    |   movel([0.036971, -1.567857, -2.417169, -0.727363, 1.570796, 1.607768],accel_mss,speed_ms,0,blend_radius_m)
    |   movel([0.032034, -1.570539, -2.414494, -0.727356, 1.570796, 1.602831],accel_mss,speed_ms,0,blend_radius_m)
    |   movel([0.033488, -1.569504, -2.415528, -0.727358, 1.570796, 1.604284],accel_mss,speed_ms,0,blend_radius_m)
    |   movel([0.034915, -1.568368, -2.416660, -0.727361, 1.570796, 1.605712],accel_mss,speed_ms,0,blend_radius_m)
    |   movel([0.036304, -1.567153, -2.417869, -0.727367, 1.570796, 1.607100],accel_mss,speed_ms,0,blend_radius_m)
    |   movel([0.037649, -1.565876, -2.419138, -0.727376, 1.570796, 1.608445],accel_mss,speed_ms,0,blend_radius_m)
    |   movel([0.040174, -1.563204, -2.421782, -0.727403, 1.570796, 1.610970],accel_mss,speed_ms,0,blend_radius_m)
    |   movel([0.042420, -1.560504, -2.424443, -0.727442, 1.570796, 1.613216],accel_mss,speed_ms,0,blend_radius_m)
    |   movel([0.044692, -1.557524, -2.427367, -0.727498, 1.570796, 1.615489],accel_mss,speed_ms,0,blend_radius_m)
    |   movel([0.046838, -1.554469, -2.430349, -0.727571, 1.570796, 1.617635],accel_mss,speed_ms,0,blend_radius_m)
    |   movel([0.047827, -1.552916, -2.431859, -0.727614, 1.570796, 1.618623],accel_mss,speed_ms,0,blend_radius_m)
    |   movel([0.048742, -1.551347, -2.433381, -0.727661, 1.570796, 1.619539],accel_mss,speed_ms,0,blend_radius_m)
    |   movel([0.049567, -1.549765, -2.434911, -0.727713, 1.570796, 1.620363],accel_mss,speed_ms,0,blend_radius_m)
    |   movel([0.050288, -1.548168, -2.436452, -0.727769, 1.570796, 1.621084],accel_mss,speed_ms,0,blend_radius_m)
    |   movel([0.050654, -1.547170, -2.437413, -0.727806, 1.570796, 1.621451],accel_mss,speed_ms,0,blend_radius_m)
    |   movel([0.050929, -1.546167, -2.438377, -0.727845, 1.570796, 1.621725],accel_mss,speed_ms,0,blend_radius_m)
    |   movel([0.051225, -1.544162, -2.440299, -0.727928, 1.570796, 1.622021],accel_mss,speed_ms,0,blend_radius_m)
    |   movel([0.051211, -1.542184, -2.442189, -0.728016, 1.570796, 1.622007],accel_mss,speed_ms,0,blend_radius_m)
    |   movel([0.050919, -1.540264, -2.444018, -0.728108, 1.570796, 1.621716],accel_mss,speed_ms,0,blend_radius_m)
    |   movel([0.050389, -1.538428, -2.445760, -0.728201, 1.570796, 1.621186],accel_mss,speed_ms,0,blend_radius_m)
    |   movel([0.049659, -1.536708, -2.447388, -0.728293, 1.570796, 1.620455],accel_mss,speed_ms,0,blend_radius_m)
    |   movel([0.048760, -1.535134, -2.448874, -0.728381, 1.570796, 1.619557],accel_mss,speed_ms,0,blend_radius_m)
    |   movel([0.047734, -1.533734, -2.450192, -0.728463, 1.570796, 1.618531],accel_mss,speed_ms,0,blend_radius_m)
    |   movel([0.046969, -1.533087, -2.450800, -0.728502, 1.570796, 1.617766],accel_mss,speed_ms,0,blend_radius_m)
    |   movel([0.046036, -1.532733, -2.451133, -0.728524, 1.570796, 1.616832],accel_mss,speed_ms,0,blend_radius_m)
    |   movel([0.044989, -1.532658, -2.451202, -0.728528, 1.570796, 1.615785],accel_mss,speed_ms,0,blend_radius_m)
    |   movel([0.043886, -1.532851, -2.451022, -0.728516, 1.570796, 1.614683],accel_mss,speed_ms,0,blend_radius_m)
    |   movel([0.042779, -1.533292, -2.450607, -0.728490, 1.570796, 1.613575],accel_mss,speed_ms,0,blend_radius_m)
    |   movel([0.041722, -1.533971, -2.449969, -0.728449, 1.570796, 1.612519],accel_mss,speed_ms,0,blend_radius_m)
    |   movel([0.040776, -1.534867, -2.449125, -0.728396, 1.570796, 1.611572],accel_mss,speed_ms,0,blend_radius_m)
    |   movel([0.039990, -1.535966, -2.448089, -0.728334, 1.570796, 1.610787],accel_mss,speed_ms,0,blend_radius_m)
    |   movel([0.038953, -1.537691, -2.446459, -0.728239, 1.570796, 1.609749],accel_mss,speed_ms,0,blend_radius_m)
    |   movel([0.037826, -1.539382, -2.444855, -0.728152, 1.570796, 1.608622],accel_mss,speed_ms,0,blend_radius_m)
    |   movel([0.036599, -1.541021, -2.443297, -0.728071, 1.570796, 1.607395],accel_mss,speed_ms,0,blend_radius_m)
    |   movel([0.035257, -1.542593, -2.441799, -0.727997, 1.570796, 1.606053],accel_mss,speed_ms,0,blend_radius_m)
    |   movel([0.033791, -1.544077, -2.440380, -0.727932, 1.570796, 1.604587],accel_mss,speed_ms,0,blend_radius_m)
    |   movel([0.032187, -1.545460, -2.439055, -0.727874, 1.570796, 1.602984],accel_mss,speed_ms,0,blend_radius_m)
    |   movel([0.030433, -1.546725, -2.437841, -0.727823, 1.570796, 1.601229],accel_mss,speed_ms,0,blend_radius_m)
    |   movel([0.028519, -1.547854, -2.436755, -0.727781, 1.570796, 1.599315],accel_mss,speed_ms,0,blend_radius_m)
    |   movel([0.027475, -1.548332, -2.436294, -0.727763, 1.570796, 1.598272],accel_mss,speed_ms,0,blend_radius_m)
    |   movel([0.026412, -1.548698, -2.435941, -0.727750, 1.570796, 1.597208],accel_mss,speed_ms,0,blend_radius_m)
    |   movel([0.024268, -1.549225, -2.435433, -0.727731, 1.570796, 1.595065],accel_mss,speed_ms,0,blend_radius_m)
    |   movel([0.022596, -1.549491, -2.435176, -0.727722, 1.570796, 1.593392],accel_mss,speed_ms,0,blend_radius_m)
    |   movel([0.021010, -1.549563, -2.435106, -0.727720, 1.570796, 1.591806],accel_mss,speed_ms,0,blend_radius_m)
    |   movel([0.019511, -1.549457, -2.435209, -0.727723, 1.570796, 1.590308],accel_mss,speed_ms,0,blend_radius_m)
    |   movel([0.018095, -1.549187, -2.435470, -0.727733, 1.570796, 1.588891],accel_mss,speed_ms,0,blend_radius_m)
    |   movel([0.016758, -1.548771, -2.435871, -0.727747, 1.570796, 1.587554],accel_mss,speed_ms,0,blend_radius_m)
    |   movel([0.015496, -1.548222, -2.436399, -0.727767, 1.570796, 1.586293],accel_mss,speed_ms,0,blend_radius_m)
    |   movel([0.014313, -1.547556, -2.437041, -0.727792, 1.570796, 1.585109],accel_mss,speed_ms,0,blend_radius_m)
    |   movel([0.013202, -1.546790, -2.437779, -0.727821, 1.570796, 1.583999],accel_mss,speed_ms,0,blend_radius_m)
    |   movel([0.012162, -1.545938, -2.438597, -0.727854, 1.570796, 1.582959],accel_mss,speed_ms,0,blend_radius_m)
    |   movel([0.011193, -1.545012, -2.439485, -0.727892, 1.570796, 1.581989],accel_mss,speed_ms,0,blend_radius_m)
    |   movel([0.009457, -1.543013, -2.441397, -0.727978, 1.570796, 1.580253],accel_mss,speed_ms,0,blend_radius_m)
    |   movel([0.007979, -1.540912, -2.443401, -0.728076, 1.570796, 1.578775],accel_mss,speed_ms,0,blend_radius_m)
    |   movel([0.006747, -1.538836, -2.445373, -0.728179, 1.570796, 1.577544],accel_mss,speed_ms,0,blend_radius_m)
    |   movel([0.005914, -1.537189, -2.446933, -0.728266, 1.570796, 1.576710],accel_mss,speed_ms,0,blend_radius_m)
    |   movel([0.005168, -1.535434, -2.448591, -0.728364, 1.570796, 1.575964],accel_mss,speed_ms,0,blend_radius_m)
    |   movel([0.004519, -1.533579, -2.450338, -0.728472, 1.570796, 1.575315],accel_mss,speed_ms,0,blend_radius_m)
    |   movel([0.003986, -1.531636, -2.452161, -0.728592, 1.570796, 1.574783],accel_mss,speed_ms,0,blend_radius_m)
    |   movel([0.003580, -1.529616, -2.454051, -0.728722, 1.570796, 1.574376],accel_mss,speed_ms,0,blend_radius_m)
    |   movel([0.003317, -1.527529, -2.455996, -0.728864, 1.570796, 1.574114],accel_mss,speed_ms,0,blend_radius_m)
    |   movel([0.003214, -1.525386, -2.457986, -0.729017, 1.570796, 1.574010],accel_mss,speed_ms,0,blend_radius_m)
    |   movel([0.003284, -1.523198, -2.460010, -0.729181, 1.570796, 1.574081],accel_mss,speed_ms,0,blend_radius_m)
    |   movel([0.003542, -1.520975, -2.462059, -0.729355, 1.570796, 1.574338],accel_mss,speed_ms,0,blend_radius_m)
    |   movel([0.004003, -1.518731, -2.464119, -0.729539, 1.570796, 1.574800],accel_mss,speed_ms,0,blend_radius_m)
    |   movel([0.004683, -1.516473, -2.466184, -0.729732, 1.570796, 1.575479],accel_mss,speed_ms,0,blend_radius_m)
    |   movel([0.005599, -1.514215, -2.468241, -0.729933, 1.570796, 1.576396],accel_mss,speed_ms,0,blend_radius_m)
    |   movel([0.006765, -1.511969, -2.470278, -0.730141, 1.570796, 1.577561],accel_mss,speed_ms,0,blend_radius_m)
    |   movel([0.008199, -1.509745, -2.472288, -0.730356, 1.570796, 1.578995],accel_mss,speed_ms,0,blend_radius_m)
    |   movel([0.009913, -1.507560, -2.474255, -0.730574, 1.570796, 1.580709],accel_mss,speed_ms,0,blend_radius_m)
    |   movel([0.011923, -1.505424, -2.476171, -0.730794, 1.570796, 1.582720],accel_mss,speed_ms,0,blend_radius_m)
    |   movel([0.012797, -1.504654, -2.476860, -0.730876, 1.570796, 1.583593],accel_mss,speed_ms,0,blend_radius_m)
    |   movel([0.013277, -1.504331, -2.477148, -0.730910, 1.570796, 1.584073],accel_mss,speed_ms,0,blend_radius_m)
    |   movel([0.013789, -1.504089, -2.477364, -0.730936, 1.570796, 1.584585],accel_mss,speed_ms,0,blend_radius_m)
    |   movel([0.014561, -1.503942, -2.477496, -0.730952, 1.570796, 1.585357],accel_mss,speed_ms,0,blend_radius_m)
    |   movel([0.015250, -1.504040, -2.477408, -0.730941, 1.570796, 1.586046],accel_mss,speed_ms,0,blend_radius_m)
    |   movel([0.015830, -1.504330, -2.477149, -0.730910, 1.570796, 1.586626],accel_mss,speed_ms,0,blend_radius_m)
    |   movel([0.016270, -1.504757, -2.476767, -0.730865, 1.570796, 1.587067],accel_mss,speed_ms,0,blend_radius_m)
    |   movel([0.016900, -1.505930, -2.475718, -0.730741, 1.570796, 1.587696],accel_mss,speed_ms,0,blend_radius_m)
    |   movel([0.017252, -1.507271, -2.474515, -0.730603, 1.570796, 1.588049],accel_mss,speed_ms,0,blend_radius_m)
    |   movel([0.017654, -1.510076, -2.471990, -0.730323, 1.570796, 1.588450],accel_mss,speed_ms,0,blend_radius_m)
    |   movel([0.017877, -1.510551, -2.471561, -0.730277, 1.570796, 1.588673],accel_mss,speed_ms,0,blend_radius_m)
    |   movel([0.018117, -1.510629, -2.471491, -0.730270, 1.570796, 1.588914],accel_mss,speed_ms,0,blend_radius_m)
    |   movel([0.018485, -1.510569, -2.471544, -0.730275, 1.570796, 1.589281],accel_mss,speed_ms,0,blend_radius_m)
    |   movel([0.019067, -1.509442, -2.472562, -0.730385, 1.570796, 1.589864],accel_mss,speed_ms,0,blend_radius_m)
    |   movel([0.019568, -1.508284, -2.473604, -0.730501, 1.570796, 1.590365],accel_mss,speed_ms,0,blend_radius_m)
    |   movel([0.019982, -1.512436, -2.469855, -0.730098, 1.570796, 1.590778],accel_mss,speed_ms,0,blend_radius_m)
    |   movel([0.020558, -1.516505, -2.466155, -0.729729, 1.570796, 1.591354],accel_mss,speed_ms,0,blend_radius_m)
    |   movel([0.021295, -1.520487, -2.462508, -0.729394, 1.570796, 1.592091],accel_mss,speed_ms,0,blend_radius_m)
    |   movel([0.022191, -1.524383, -2.458915, -0.729091, 1.570796, 1.592987],accel_mss,speed_ms,0,blend_radius_m)
    |   movel([0.022649, -1.526045, -2.457375, -0.728969, 1.570796, 1.593445],accel_mss,speed_ms,0,blend_radius_m)
    |   movel([0.023296, -1.527701, -2.455836, -0.728852, 1.570796, 1.594092],accel_mss,speed_ms,0,blend_radius_m)
    |   movel([0.023724, -1.528467, -2.455122, -0.728800, 1.570796, 1.594520],accel_mss,speed_ms,0,blend_radius_m)
    |   movel([0.024238, -1.529159, -2.454478, -0.728753, 1.570796, 1.595035],accel_mss,speed_ms,0,blend_radius_m)
    |   movel([0.024855, -1.529751, -2.453924, -0.728713, 1.570796, 1.595651],accel_mss,speed_ms,0,blend_radius_m)
    |   movel([0.025587, -1.530219, -2.453487, -0.728683, 1.570796, 1.596384],accel_mss,speed_ms,0,blend_radius_m)
    |   movel([0.026170, -1.530452, -2.453270, -0.728668, 1.570796, 1.596966],accel_mss,speed_ms,0,blend_radius_m)
    |   movel([0.027457, -1.530642, -2.453092, -0.728655, 1.570796, 1.598253],accel_mss,speed_ms,0,blend_radius_m)
    |   movel([0.028149, -1.530613, -2.453119, -0.728657, 1.570796, 1.598945],accel_mss,speed_ms,0,blend_radius_m)
    |   movel([0.029599, -1.530339, -2.453375, -0.728675, 1.570796, 1.600395],accel_mss,speed_ms,0,blend_radius_m)
    |   movel([0.031098, -1.529820, -2.453860, -0.728709, 1.570796, 1.601894],accel_mss,speed_ms,0,blend_radius_m)
    |   movel([0.032596, -1.529109, -2.454524, -0.728756, 1.570796, 1.603392],accel_mss,speed_ms,0,blend_radius_m)
    |   movel([0.034042, -1.528253, -2.455322, -0.728814, 1.570796, 1.604839],accel_mss,speed_ms,0,blend_radius_m)
    |   movel([0.035389, -1.527306, -2.456203, -0.728880, 1.570796, 1.606186],accel_mss,speed_ms,0,blend_radius_m)
    |   movel([0.036582, -1.526318, -2.457121, -0.728950, 1.570796, 1.607378],accel_mss,speed_ms,0,blend_radius_m)
    |   speed_ms = 0.005
    |   movel([0.036582, -1.518669, -2.453733, -0.739987, 1.570796, 1.607378],accel_mss,speed_ms,0,blend_radius_m)
    |   speed_ms = 0.040
    |   movel([0.029707, -1.520999, -2.451592, -0.739798, 1.570796, 1.600503],accel_mss,speed_ms,0,blend_radius_m)
    |   speed_ms = 0.005
    |   movel([0.029707, -1.528629, -2.454972, -0.728789, 1.570796, 1.600503],accel_mss,speed_ms,0,blend_radius_m)
    |   speed_ms = 0.025
    |   movel([0.030662, -1.527790, -2.455753, -0.728846, 1.570796, 1.601458],accel_mss,speed_ms,0,blend_radius_m)
    |   movel([0.032483, -1.525887, -2.457521, -0.728981, 1.570796, 1.603279],accel_mss,speed_ms,0,blend_radius_m)
    |   movel([0.033332, -1.524844, -2.458488, -0.729057, 1.570796, 1.604128],accel_mss,speed_ms,0,blend_radius_m)
    |   movel([0.034867, -1.522630, -2.460534, -0.729225, 1.570796, 1.605663],accel_mss,speed_ms,0,blend_radius_m)
    |   movel([0.036139, -1.520315, -2.462665, -0.729408, 1.570796, 1.606935],accel_mss,speed_ms,0,blend_radius_m)
    |   movel([0.036655, -1.519150, -2.463735, -0.729504, 1.570796, 1.607451],accel_mss,speed_ms,0,blend_radius_m)
    |   movel([0.037080, -1.517990, -2.464798, -0.729601, 1.570796, 1.607876],accel_mss,speed_ms,0,blend_radius_m)
    |   movel([0.037625, -1.515742, -2.466851, -0.729796, 1.570796, 1.608421],accel_mss,speed_ms,0,blend_radius_m)
    |   movel([0.037730, -1.514673, -2.467824, -0.729892, 1.570796, 1.608527],accel_mss,speed_ms,0,blend_radius_m)
    |   movel([0.037711, -1.513660, -2.468745, -0.729984, 1.570796, 1.608507],accel_mss,speed_ms,0,blend_radius_m)
    |   movel([0.037562, -1.512711, -2.469606, -0.730072, 1.570796, 1.608358],accel_mss,speed_ms,0,blend_radius_m)
    |   movel([0.037272, -1.511838, -2.470397, -0.730154, 1.570796, 1.608069],accel_mss,speed_ms,0,blend_radius_m)
    |   movel([0.036758, -1.510843, -2.471297, -0.730249, 1.570796, 1.607554],accel_mss,speed_ms,0,blend_radius_m)
    |   movel([0.036113, -1.509942, -2.472111, -0.730336, 1.570796, 1.606909],accel_mss,speed_ms,0,blend_radius_m)
    |   movel([0.035329, -1.509166, -2.472810, -0.730413, 1.570796, 1.606125],accel_mss,speed_ms,0,blend_radius_m)
    |   movel([0.034399, -1.508552, -2.473363, -0.730474, 1.570796, 1.605195],accel_mss,speed_ms,0,blend_radius_m)
    |   movel([0.033317, -1.508132, -2.473741, -0.730516, 1.570796, 1.604113],accel_mss,speed_ms,0,blend_radius_m)
    |   movel([0.032079, -1.507942, -2.473912, -0.730535, 1.570796, 1.602875],accel_mss,speed_ms,0,blend_radius_m)
    |   movel([0.030678, -1.508015, -2.473846, -0.730528, 1.570796, 1.601475],accel_mss,speed_ms,0,blend_radius_m)
    |   movel([0.029111, -1.508381, -2.473517, -0.730491, 1.570796, 1.599907],accel_mss,speed_ms,0,blend_radius_m)
    |   movel([0.028034, -1.508807, -2.473134, -0.730448, 1.570796, 1.598830],accel_mss,speed_ms,0,blend_radius_m)
    |   movel([0.026989, -1.509378, -2.472620, -0.730392, 1.570796, 1.597785],accel_mss,speed_ms,0,blend_radius_m)
    |   movel([0.026011, -1.510066, -2.471999, -0.730324, 1.570796, 1.596808],accel_mss,speed_ms,0,blend_radius_m)
    |   movel([0.025131, -1.510848, -2.471292, -0.730248, 1.570796, 1.595927],accel_mss,speed_ms,0,blend_radius_m)
    |   movel([0.024378, -1.511699, -2.470523, -0.730167, 1.570796, 1.595174],accel_mss,speed_ms,0,blend_radius_m)
    |   movel([0.023782, -1.512594, -2.469713, -0.730083, 1.570796, 1.594578],accel_mss,speed_ms,0,blend_radius_m)
    |   movel([0.023377, -1.513506, -2.468884, -0.729998, 1.570796, 1.594173],accel_mss,speed_ms,0,blend_radius_m)
    |   movel([0.023187, -1.514415, -2.468059, -0.729915, 1.570796, 1.593984],accel_mss,speed_ms,0,blend_radius_m)
    |   speed_ms = 0.005
    |   movel([0.023187, -1.506669, -2.464625, -0.741095, 1.570796, 1.593984],accel_mss,speed_ms,0,blend_radius_m)
    |   speed_ms = 0.040
    |   # Splitting Linear movement in 2 (instruction 399: MoveL 378)
    |   movel([0.051290, -1.516388, -2.455821, -0.740180, 1.570796, 1.622087],accel_mss,speed_ms,0,blend_radius_m)
    |   movel([0.078430, -1.526900, -2.446130, -0.739359, 1.570796, 1.649227],accel_mss,speed_ms,0,blend_radius_m)
    |   speed_ms = 0.005
    |   movel([0.078430, -1.534483, -2.449487, -0.728419, 1.570796, 1.649227],accel_mss,speed_ms,0,blend_radius_m)
    |   speed_ms = 0.025
    |   movel([0.077845, -1.539171, -2.445055, -0.728162, 1.570796, 1.648641],accel_mss,speed_ms,0,blend_radius_m)
    |   movel([0.077355, -1.541529, -2.442814, -0.728047, 1.570796, 1.648151],accel_mss,speed_ms,0,blend_radius_m)
    |   movel([0.076991, -1.542730, -2.441668, -0.727991, 1.570796, 1.647787],accel_mss,speed_ms,0,blend_radius_m)
    |   movel([0.076521, -1.543950, -2.440502, -0.727937, 1.570796, 1.647317],accel_mss,speed_ms,0,blend_radius_m)
    |   movel([0.075883, -1.545241, -2.439265, -0.727883, 1.570796, 1.646679],accel_mss,speed_ms,0,blend_radius_m)
    |   movel([0.075474, -1.545865, -2.438667, -0.727857, 1.570796, 1.646270],accel_mss,speed_ms,0,blend_radius_m)
    |   movel([0.074975, -1.546457, -2.438098, -0.727834, 1.570796, 1.645772],accel_mss,speed_ms,0,blend_radius_m)
    |   movel([0.074917, -1.545380, -2.439132, -0.727877, 1.570796, 1.645713],accel_mss,speed_ms,0,blend_radius_m)
    |   movel([0.074651, -1.544385, -2.440086, -0.727919, 1.570796, 1.645447],accel_mss,speed_ms,0,blend_radius_m)
    |   movel([0.074441, -1.544113, -2.440346, -0.727930, 1.570796, 1.645237],accel_mss,speed_ms,0,blend_radius_m)
    |   movel([0.074235, -1.544095, -2.440363, -0.727931, 1.570796, 1.645031],accel_mss,speed_ms,0,blend_radius_m)
    |   movel([0.074002, -1.544166, -2.440295, -0.727928, 1.570796, 1.644799],accel_mss,speed_ms,0,blend_radius_m)
    |   movel([0.073546, -1.544468, -2.440006, -0.727915, 1.570796, 1.644342],accel_mss,speed_ms,0,blend_radius_m)
    |   movel([0.072920, -1.545089, -2.439411, -0.727889, 1.570796, 1.643716],accel_mss,speed_ms,0,blend_radius_m)
    |   movel([0.072434, -1.545739, -2.438788, -0.727862, 1.570796, 1.643230],accel_mss,speed_ms,0,blend_radius_m)
    |   movel([0.072061, -1.546408, -2.438145, -0.727836, 1.570796, 1.642857],accel_mss,speed_ms,0,blend_radius_m)
    |   movel([0.071777, -1.547091, -2.437489, -0.727809, 1.570796, 1.642573],accel_mss,speed_ms,0,blend_radius_m)
    |   movel([0.070981, -1.549850, -2.434829, -0.727710, 1.570796, 1.641778],accel_mss,speed_ms,0,blend_radius_m)
    |   movel([0.070413, -1.551470, -2.433262, -0.727657, 1.570796, 1.641209],accel_mss,speed_ms,0,blend_radius_m)
    |   movel([0.069717, -1.553085, -2.431695, -0.727609, 1.570796, 1.640513],accel_mss,speed_ms,0,blend_radius_m)
    |   movel([0.068858, -1.554681, -2.430142, -0.727566, 1.570796, 1.639655],accel_mss,speed_ms,0,blend_radius_m)
    |   movel([0.067805, -1.556238, -2.428624, -0.727527, 1.570796, 1.638601],accel_mss,speed_ms,0,blend_radius_m)
    |   movel([0.068063, -1.554979, -2.429852, -0.727558, 1.570796, 1.638860],accel_mss,speed_ms,0,blend_radius_m)
    |   movel([0.067978, -1.553800, -2.431000, -0.727589, 1.570796, 1.638774],accel_mss,speed_ms,0,blend_radius_m)
    |   movel([0.067880, -1.553531, -2.431261, -0.727597, 1.570796, 1.638676],accel_mss,speed_ms,0,blend_radius_m)
    |   movel([0.067664, -1.553353, -2.431434, -0.727602, 1.570796, 1.638460],accel_mss,speed_ms,0,blend_radius_m)
    |   movel([0.067395, -1.553343, -2.431444, -0.727602, 1.570796, 1.638191],accel_mss,speed_ms,0,blend_radius_m)
    |   movel([0.067096, -1.553445, -2.431345, -0.727599, 1.570796, 1.637893],accel_mss,speed_ms,0,blend_radius_m)
    |   movel([0.066527, -1.553838, -2.430963, -0.727588, 1.570796, 1.637323],accel_mss,speed_ms,0,blend_radius_m)
    |   movel([0.065929, -1.554444, -2.430373, -0.727572, 1.570796, 1.636725],accel_mss,speed_ms,0,blend_radius_m)
    |   movel([0.065425, -1.555097, -2.429737, -0.727555, 1.570796, 1.636222],accel_mss,speed_ms,0,blend_radius_m)
    |   movel([0.064630, -1.556488, -2.428379, -0.727521, 1.570796, 1.635426],accel_mss,speed_ms,0,blend_radius_m)
    |   movel([0.063348, -1.559296, -2.425630, -0.727463, 1.570796, 1.634145],accel_mss,speed_ms,0,blend_radius_m)
    |   movel([0.062488, -1.560840, -2.424112, -0.727436, 1.570796, 1.633284],accel_mss,speed_ms,0,blend_radius_m)
    |   movel([0.061504, -1.562357, -2.422618, -0.727414, 1.570796, 1.632300],accel_mss,speed_ms,0,blend_radius_m)
    |   movel([0.060367, -1.563818, -2.421175, -0.727396, 1.570796, 1.631163],accel_mss,speed_ms,0,blend_radius_m)
    |   movel([0.059049, -1.565195, -2.419812, -0.727382, 1.570796, 1.629845],accel_mss,speed_ms,0,blend_radius_m)
    |   movel([0.059292, -1.564503, -2.420497, -0.727388, 1.570796, 1.630088],accel_mss,speed_ms,0,blend_radius_m)
    |   movel([0.059487, -1.563157, -2.421829, -0.727403, 1.570796, 1.630284],accel_mss,speed_ms,0,blend_radius_m)
    |   movel([0.059436, -1.562520, -2.422457, -0.727412, 1.570796, 1.630232],accel_mss,speed_ms,0,blend_radius_m)
    |   movel([0.059334, -1.562256, -2.422718, -0.727415, 1.570796, 1.630130],accel_mss,speed_ms,0,blend_radius_m)
    |   movel([0.059075, -1.562157, -2.422815, -0.727416, 1.570796, 1.629871],accel_mss,speed_ms,0,blend_radius_m)
    |   movel([0.058716, -1.562339, -2.422636, -0.727414, 1.570796, 1.629513],accel_mss,speed_ms,0,blend_radius_m)
    |   movel([0.057925, -1.562984, -2.422000, -0.727405, 1.570796, 1.628722],accel_mss,speed_ms,0,blend_radius_m)
    |   movel([0.057246, -1.563664, -2.421327, -0.727397, 1.570796, 1.628042],accel_mss,speed_ms,0,blend_radius_m)
    |   movel([0.056090, -1.565100, -2.419907, -0.727382, 1.570796, 1.626886],accel_mss,speed_ms,0,blend_radius_m)
    |   movel([0.054983, -1.566564, -2.418454, -0.727371, 1.570796, 1.625780],accel_mss,speed_ms,0,blend_radius_m)
    |   movel([0.054365, -1.567285, -2.417738, -0.727366, 1.570796, 1.625161],accel_mss,speed_ms,0,blend_radius_m)
    |   movel([0.053658, -1.567985, -2.417041, -0.727363, 1.570796, 1.624454],accel_mss,speed_ms,0,blend_radius_m)
    |   movel([0.051800, -1.569572, -2.415460, -0.727357, 1.570796, 1.622596],accel_mss,speed_ms,0,blend_radius_m)
    |   movel([0.049863, -1.571079, -2.413954, -0.727356, 1.570796, 1.620660],accel_mss,speed_ms,0,blend_radius_m)
    |   movel([0.047871, -1.572512, -2.412518, -0.727359, 1.570796, 1.618667],accel_mss,speed_ms,0,blend_radius_m)
    |   movel([0.045837, -1.573884, -2.411141, -0.727364, 1.570796, 1.616634],accel_mss,speed_ms,0,blend_radius_m)
    |   speed_ms = 0.005
    |   movel([0.045837, -1.566622, -2.407929, -0.737838, 1.570796, 1.616634],accel_mss,speed_ms,0,blend_radius_m)
    |   speed_ms = 0.040
    |   movel([0.029341, -1.549189, -2.425003, -0.738197, 1.570796, 1.600137],accel_mss,speed_ms,0,blend_radius_m)
    |   speed_ms = 0.005
    |   movel([0.029341, -1.556592, -2.428278, -0.727519, 1.570796, 1.600137],accel_mss,speed_ms,0,blend_radius_m)
    |   speed_ms = 0.025
    |   movel([0.029967, -1.556056, -2.428801, -0.727531, 1.570796, 1.600763],accel_mss,speed_ms,0,blend_radius_m)
    |   movel([0.030522, -1.555448, -2.429395, -0.727546, 1.570796, 1.601318],accel_mss,speed_ms,0,blend_radius_m)
    |   movel([0.031512, -1.554098, -2.430710, -0.727581, 1.570796, 1.602308],accel_mss,speed_ms,0,blend_radius_m)
    |   movel([0.032486, -1.552713, -2.432056, -0.727620, 1.570796, 1.603282],accel_mss,speed_ms,0,blend_radius_m)
    |   movel([0.033024, -1.552059, -2.432690, -0.727639, 1.570796, 1.603820],accel_mss,speed_ms,0,blend_radius_m)
    |   movel([0.033625, -1.551460, -2.433271, -0.727658, 1.570796, 1.604422],accel_mss,speed_ms,0,blend_radius_m)
    |   movel([0.034109, -1.551081, -2.433639, -0.727670, 1.570796, 1.604905],accel_mss,speed_ms,0,blend_radius_m)
    |   movel([0.034514, -1.550857, -2.433855, -0.727677, 1.570796, 1.605310],accel_mss,speed_ms,0,blend_radius_m)
    |   movel([0.034846, -1.550772, -2.433938, -0.727680, 1.570796, 1.605642],accel_mss,speed_ms,0,blend_radius_m)
    |   movel([0.035114, -1.550807, -2.433904, -0.727678, 1.570796, 1.605910],accel_mss,speed_ms,0,blend_radius_m)
    |   movel([0.035476, -1.551181, -2.433541, -0.727666, 1.570796, 1.606273],accel_mss,speed_ms,0,blend_radius_m)
    |   movel([0.035654, -1.551846, -2.432897, -0.727646, 1.570796, 1.606451],accel_mss,speed_ms,0,blend_radius_m)
    |   movel([0.035652, -1.553528, -2.431265, -0.727597, 1.570796, 1.606449],accel_mss,speed_ms,0,blend_radius_m)
    |   movel([0.035520, -1.554807, -2.430019, -0.727562, 1.570796, 1.606317],accel_mss,speed_ms,0,blend_radius_m)
    |   movel([0.036607, -1.553451, -2.431340, -0.727599, 1.570796, 1.607403],accel_mss,speed_ms,0,blend_radius_m)
    |   movel([0.037417, -1.552109, -2.432642, -0.727638, 1.570796, 1.608213],accel_mss,speed_ms,0,blend_radius_m)
    |   movel([0.038022, -1.550775, -2.433935, -0.727679, 1.570796, 1.608818],accel_mss,speed_ms,0,blend_radius_m)
    |   movel([0.038487, -1.549443, -2.435222, -0.727724, 1.570796, 1.609283],accel_mss,speed_ms,0,blend_radius_m)
    |   movel([0.039732, -1.545392, -2.439121, -0.727876, 1.570796, 1.610528],accel_mss,speed_ms,0,blend_radius_m)
    |   movel([0.040325, -1.544001, -2.440453, -0.727935, 1.570796, 1.611121],accel_mss,speed_ms,0,blend_radius_m)
    |   movel([0.040666, -1.543456, -2.440974, -0.727959, 1.570796, 1.611462],accel_mss,speed_ms,0,blend_radius_m)
    |   movel([0.041027, -1.543133, -2.441283, -0.727973, 1.570796, 1.611823],accel_mss,speed_ms,0,blend_radius_m)
    |   movel([0.041393, -1.542997, -2.441413, -0.727979, 1.570796, 1.612189],accel_mss,speed_ms,0,blend_radius_m)
    |   movel([0.041747, -1.543018, -2.441393, -0.727978, 1.570796, 1.612544],accel_mss,speed_ms,0,blend_radius_m)
    |   movel([0.042077, -1.543160, -2.441257, -0.727972, 1.570796, 1.612873],accel_mss,speed_ms,0,blend_radius_m)
    |   movel([0.042363, -1.543391, -2.441036, -0.727962, 1.570796, 1.613159],accel_mss,speed_ms,0,blend_radius_m)
    |   movel([0.042751, -1.543986, -2.440468, -0.727936, 1.570796, 1.613547],accel_mss,speed_ms,0,blend_radius_m)
    |   movel([0.042858, -1.544696, -2.439788, -0.727905, 1.570796, 1.613655],accel_mss,speed_ms,0,blend_radius_m)
    |   movel([0.042815, -1.545644, -2.438879, -0.727866, 1.570796, 1.613612],accel_mss,speed_ms,0,blend_radius_m)
    |   movel([0.042602, -1.547416, -2.437176, -0.727797, 1.570796, 1.613398],accel_mss,speed_ms,0,blend_radius_m)
    |   movel([0.043636, -1.544669, -2.439814, -0.727907, 1.570796, 1.614432],accel_mss,speed_ms,0,blend_radius_m)
    |   movel([0.044012, -1.543300, -2.441124, -0.727966, 1.570796, 1.614808],accel_mss,speed_ms,0,blend_radius_m)
    |   movel([0.044476, -1.540592, -2.443706, -0.728092, 1.570796, 1.615272],accel_mss,speed_ms,0,blend_radius_m)
    |   movel([0.044559, -1.539266, -2.444965, -0.728157, 1.570796, 1.615356],accel_mss,speed_ms,0,blend_radius_m)
    |   movel([0.044427, -1.536697, -2.447399, -0.728293, 1.570796, 1.615223],accel_mss,speed_ms,0,blend_radius_m)
    |   speed_ms = 0.005
    |   movel([0.044427, -1.529132, -2.444050, -0.739207, 1.570796, 1.615223],accel_mss,speed_ms,0,blend_radius_m)
    |   speed_ms = 0.040
    |   movel([0.034396, -1.539639, -2.434152, -0.738598, 1.570796, 1.605192],accel_mss,speed_ms,0,blend_radius_m)
    |   speed_ms = 0.005
    |   movel([0.034396, -1.547119, -2.437462, -0.727808, 1.570796, 1.605192],accel_mss,speed_ms,0,blend_radius_m)
    |   speed_ms = 0.025
    |   movel([0.033124, -1.548649, -2.435989, -0.727752, 1.570796, 1.603921],accel_mss,speed_ms,0,blend_radius_m)
    |   movel([0.031967, -1.550220, -2.434471, -0.727698, 1.570796, 1.602764],accel_mss,speed_ms,0,blend_radius_m)
    |   movel([0.029723, -1.553380, -2.431408, -0.727601, 1.570796, 1.600519],accel_mss,speed_ms,0,blend_radius_m)
    |   movel([0.028483, -1.554925, -2.429905, -0.727559, 1.570796, 1.599279],accel_mss,speed_ms,0,blend_radius_m)
    |   movel([0.027098, -1.556390, -2.428475, -0.727524, 1.570796, 1.597895],accel_mss,speed_ms,0,blend_radius_m)
    |   movel([0.025552, -1.557703, -2.427192, -0.727495, 1.570796, 1.596348],accel_mss,speed_ms,0,blend_radius_m)
    |   movel([0.024714, -1.558279, -2.426628, -0.727483, 1.570796, 1.595510],accel_mss,speed_ms,0,blend_radius_m)
    |   movel([0.023830, -1.558789, -2.426128, -0.727473, 1.570796, 1.594627],accel_mss,speed_ms,0,blend_radius_m)
    |   movel([0.024473, -1.558300, -2.426607, -0.727482, 1.570796, 1.595270],accel_mss,speed_ms,0,blend_radius_m)
    |   movel([0.025137, -1.557542, -2.427349, -0.727498, 1.570796, 1.595934],accel_mss,speed_ms,0,blend_radius_m)
    |   movel([0.025747, -1.556626, -2.428245, -0.727518, 1.570796, 1.596543],accel_mss,speed_ms,0,blend_radius_m)
    |   movel([0.026215, -1.555667, -2.429182, -0.727541, 1.570796, 1.597012],accel_mss,speed_ms,0,blend_radius_m)
    |   movel([0.026464, -1.554775, -2.430050, -0.727563, 1.570796, 1.597260],accel_mss,speed_ms,0,blend_radius_m)
    |   movel([0.026478, -1.554394, -2.430422, -0.727573, 1.570796, 1.597275],accel_mss,speed_ms,0,blend_radius_m)
    |   movel([0.026408, -1.554072, -2.430735, -0.727582, 1.570796, 1.597204],accel_mss,speed_ms,0,blend_radius_m)
    |   movel([0.026242, -1.553823, -2.430977, -0.727589, 1.570796, 1.597038],accel_mss,speed_ms,0,blend_radius_m)
    |   movel([0.025967, -1.553666, -2.431130, -0.727593, 1.570796, 1.596764],accel_mss,speed_ms,0,blend_radius_m)
    |   movel([0.025578, -1.553610, -2.431184, -0.727594, 1.570796, 1.596374],accel_mss,speed_ms,0,blend_radius_m)
    |   movel([0.025059, -1.553673, -2.431123, -0.727593, 1.570796, 1.595856],accel_mss,speed_ms,0,blend_radius_m)
    |   movel([0.024231, -1.554003, -2.430802, -0.727584, 1.570796, 1.595027],accel_mss,speed_ms,0,blend_radius_m)
    |   movel([0.020833, -1.556030, -2.428827, -0.727532, 1.570796, 1.591629],accel_mss,speed_ms,0,blend_radius_m)
    |   movel([0.019373, -1.556765, -2.428109, -0.727515, 1.570796, 1.590169],accel_mss,speed_ms,0,blend_radius_m)
    |   movel([0.017870, -1.557410, -2.427478, -0.727501, 1.570796, 1.588666],accel_mss,speed_ms,0,blend_radius_m)
    |   movel([0.016371, -1.557921, -2.426978, -0.727490, 1.570796, 1.587168],accel_mss,speed_ms,0,blend_radius_m)
    |   movel([0.014924, -1.558247, -2.426658, -0.727483, 1.570796, 1.585720],accel_mss,speed_ms,0,blend_radius_m)
    |   movel([0.013571, -1.558343, -2.426564, -0.727481, 1.570796, 1.584368],accel_mss,speed_ms,0,blend_radius_m)
    |   movel([0.012362, -1.558158, -2.426746, -0.727485, 1.570796, 1.583159],accel_mss,speed_ms,0,blend_radius_m)
    |   movel([0.012749, -1.558163, -2.426741, -0.727485, 1.570796, 1.583545],accel_mss,speed_ms,0,blend_radius_m)
    |   movel([0.013255, -1.558014, -2.426887, -0.727488, 1.570796, 1.584051],accel_mss,speed_ms,0,blend_radius_m)
    |   movel([0.014465, -1.557405, -2.427483, -0.727501, 1.570796, 1.585262],accel_mss,speed_ms,0,blend_radius_m)
    |   movel([0.015650, -1.556628, -2.428243, -0.727518, 1.570796, 1.586446],accel_mss,speed_ms,0,blend_radius_m)
    |   movel([0.016463, -1.555984, -2.428872, -0.727533, 1.570796, 1.587259],accel_mss,speed_ms,0,blend_radius_m)
    |   movel([0.016937, -1.555461, -2.429382, -0.727546, 1.570796, 1.587734],accel_mss,speed_ms,0,blend_radius_m)
    |   movel([0.017112, -1.555085, -2.429748, -0.727555, 1.570796, 1.587908],accel_mss,speed_ms,0,blend_radius_m)
    |   movel([0.017034, -1.554834, -2.429993, -0.727562, 1.570796, 1.587830],accel_mss,speed_ms,0,blend_radius_m)
    |   movel([0.016759, -1.554686, -2.430138, -0.727566, 1.570796, 1.587555],accel_mss,speed_ms,0,blend_radius_m)
    |   movel([0.015833, -1.554607, -2.430214, -0.727568, 1.570796, 1.586629],accel_mss,speed_ms,0,blend_radius_m)
    |   movel([0.014762, -1.554673, -2.430150, -0.727566, 1.570796, 1.585558],accel_mss,speed_ms,0,blend_radius_m)
    |   movel([0.012326, -1.554819, -2.430008, -0.727562, 1.570796, 1.583122],accel_mss,speed_ms,0,blend_radius_m)
    |   movel([0.009899, -1.554777, -2.430049, -0.727563, 1.570796, 1.580695],accel_mss,speed_ms,0,blend_radius_m)
    |   movel([0.008753, -1.554631, -2.430191, -0.727567, 1.570796, 1.579550],accel_mss,speed_ms,0,blend_radius_m)
    |   movel([0.007687, -1.554372, -2.430443, -0.727574, 1.570796, 1.578484],accel_mss,speed_ms,0,blend_radius_m)
    |   movel([0.006727, -1.553977, -2.430827, -0.727584, 1.570796, 1.577523],accel_mss,speed_ms,0,blend_radius_m)
    |   movel([0.005899, -1.553426, -2.431364, -0.727600, 1.570796, 1.576696],accel_mss,speed_ms,0,blend_radius_m)
    |   movel([0.007352, -1.553330, -2.431457, -0.727602, 1.570796, 1.578149],accel_mss,speed_ms,0,blend_radius_m)
    |   movel([0.008148, -1.553123, -2.431658, -0.727608, 1.570796, 1.578944],accel_mss,speed_ms,0,blend_radius_m)
    |   movel([0.008500, -1.552950, -2.431826, -0.727613, 1.570796, 1.579296],accel_mss,speed_ms,0,blend_radius_m)
    |   movel([0.008800, -1.552716, -2.432053, -0.727620, 1.570796, 1.579597],accel_mss,speed_ms,0,blend_radius_m)
    |   movel([0.008923, -1.552515, -2.432248, -0.727626, 1.570796, 1.579719],accel_mss,speed_ms,0,blend_radius_m)
    |   movel([0.008905, -1.552303, -2.432454, -0.727632, 1.570796, 1.579701],accel_mss,speed_ms,0,blend_radius_m)
    |   movel([0.008524, -1.551863, -2.432881, -0.727645, 1.570796, 1.579320],accel_mss,speed_ms,0,blend_radius_m)
    |   movel([0.007787, -1.551416, -2.433314, -0.727659, 1.570796, 1.578583],accel_mss,speed_ms,0,blend_radius_m)
    |   movel([0.006830, -1.550983, -2.433734, -0.727673, 1.570796, 1.577626],accel_mss,speed_ms,0,blend_radius_m)
    |   movel([0.003478, -1.549785, -2.434892, -0.727712, 1.570796, 1.574275],accel_mss,speed_ms,0,blend_radius_m)
    |   movel([0.002266, -1.549172, -2.435484, -0.727733, 1.570796, 1.573062],accel_mss,speed_ms,0,blend_radius_m)
    |   movel([0.001172, -1.548431, -2.436199, -0.727760, 1.570796, 1.571968],accel_mss,speed_ms,0,blend_radius_m)
    |   movel([0.000270, -1.547536, -2.437061, -0.727792, 1.570796, 1.571066],accel_mss,speed_ms,0,blend_radius_m)
    |   movel([-0.000379, -1.546461, -2.438095, -0.727834, 1.570796, 1.570417],accel_mss,speed_ms,0,blend_radius_m)
    |   movel([0.000737, -1.547091, -2.437489, -0.727809, 1.570796, 1.571534],accel_mss,speed_ms,0,blend_radius_m)
    |   movel([0.001435, -1.547315, -2.437273, -0.727801, 1.570796, 1.572231],accel_mss,speed_ms,0,blend_radius_m)
    |   movel([0.002114, -1.547316, -2.437272, -0.727801, 1.570796, 1.572911],accel_mss,speed_ms,0,blend_radius_m)
    |   movel([0.002763, -1.547052, -2.437526, -0.727811, 1.570796, 1.573560],accel_mss,speed_ms,0,blend_radius_m)
    |   movel([0.003154, -1.546657, -2.437906, -0.727826, 1.570796, 1.573950],accel_mss,speed_ms,0,blend_radius_m)
    |   movel([0.003271, -1.546193, -2.438352, -0.727844, 1.570796, 1.574067],accel_mss,speed_ms,0,blend_radius_m)
    |   movel([0.003102, -1.545720, -2.438806, -0.727863, 1.570796, 1.573898],accel_mss,speed_ms,0,blend_radius_m)
    |   movel([0.001694, -1.543429, -2.441000, -0.727960, 1.570796, 1.572491],accel_mss,speed_ms,0,blend_radius_m)
    |   movel([0.000629, -1.541006, -2.443311, -0.728071, 1.570796, 1.571425],accel_mss,speed_ms,0,blend_radius_m)
    |   movel([0.000249, -1.539716, -2.444538, -0.728135, 1.570796, 1.571046],accel_mss,speed_ms,0,blend_radius_m)
    |   movel([-0.000017, -1.538359, -2.445826, -0.728204, 1.570796, 1.570780],accel_mss,speed_ms,0,blend_radius_m)
    |   movel([-0.000159, -1.536921, -2.447187, -0.728281, 1.570796, 1.570638],accel_mss,speed_ms,0,blend_radius_m)
    |   movel([-0.000167, -1.535393, -2.448630, -0.728366, 1.570796, 1.570629],accel_mss,speed_ms,0,blend_radius_m)
    |   speed_ms = 0.005
    |   movel([-0.000167, -1.527817, -2.445276, -0.739295, 1.570796, 1.570629],accel_mss,speed_ms,0,blend_radius_m)
    |   speed_ms = 0.040
    |   movel([-0.022466, -1.518241, -2.454125, -0.740023, 1.570796, 1.548330],accel_mss,speed_ms,0,blend_radius_m)
    |   speed_ms = 0.005
    |   movel([-0.022466, -1.525894, -2.457515, -0.728980, 1.570796, 1.548330],accel_mss,speed_ms,0,blend_radius_m)
    |   speed_ms = 0.025
    |   movel([-0.020597, -1.523608, -2.459632, -0.729150, 1.570796, 1.550199],accel_mss,speed_ms,0,blend_radius_m)
    |   movel([-0.018803, -1.521289, -2.461770, -0.729330, 1.570796, 1.551993],accel_mss,speed_ms,0,blend_radius_m)
    |   movel([-0.015402, -1.516544, -2.466119, -0.729726, 1.570796, 1.555394],accel_mss,speed_ms,0,blend_radius_m)
    |   movel([-0.012257, -1.511675, -2.470545, -0.730169, 1.570796, 1.558539],accel_mss,speed_ms,0,blend_radius_m)
    |   movel([-0.009374, -1.506698, -2.475029, -0.730662, 1.570796, 1.561423],accel_mss,speed_ms,0,blend_radius_m)
    |   movel([-0.006758, -1.501628, -2.479557, -0.731204, 1.570796, 1.564039],accel_mss,speed_ms,0,blend_radius_m)
    |   movel([-0.004417, -1.496483, -2.484110, -0.731796, 1.570796, 1.566379],accel_mss,speed_ms,0,blend_radius_m)
    |   movel([-0.002357, -1.491285, -2.488667, -0.732437, 1.570796, 1.568439],accel_mss,speed_ms,0,blend_radius_m)
    |   movel([-0.000586, -1.486048, -2.493215, -0.733125, 1.570796, 1.570210],accel_mss,speed_ms,0,blend_radius_m)
    |   movel([0.000887, -1.480798, -2.497732, -0.733859, 1.570796, 1.571683],accel_mss,speed_ms,0,blend_radius_m)
    |   movel([0.002055, -1.475554, -2.502200, -0.734635, 1.570796, 1.572851],accel_mss,speed_ms,0,blend_radius_m)
    |   movel([0.002907, -1.470339, -2.506601, -0.735450, 1.570796, 1.573704],accel_mss,speed_ms,0,blend_radius_m)
    |   movel([0.003433, -1.465176, -2.510915, -0.736298, 1.570796, 1.574229],accel_mss,speed_ms,0,blend_radius_m)
    |   movel([0.003629, -1.460086, -2.515128, -0.737175, 1.570796, 1.574425],accel_mss,speed_ms,0,blend_radius_m)
    |   movel([0.003478, -1.455098, -2.519218, -0.738073, 1.570796, 1.574274],accel_mss,speed_ms,0,blend_radius_m)
    |   movel([0.002975, -1.450238, -2.523165, -0.738986, 1.570796, 1.573771],accel_mss,speed_ms,0,blend_radius_m)
    |   movel([0.001663, -1.443176, -2.528837, -0.740376, 1.570796, 1.572460],accel_mss,speed_ms,0,blend_radius_m)
    |   movel([0.001633, -1.441931, -2.529829, -0.740629, 1.570796, 1.572429],accel_mss,speed_ms,0,blend_radius_m)
    |   movel([0.001847, -1.440618, -2.530872, -0.740898, 1.570796, 1.572643],accel_mss,speed_ms,0,blend_radius_m)
    |   movel([0.002491, -1.438763, -2.532343, -0.741284, 1.570796, 1.573287],accel_mss,speed_ms,0,blend_radius_m)
    |   movel([0.003293, -1.437317, -2.533484, -0.741587, 1.570796, 1.574089],accel_mss,speed_ms,0,blend_radius_m)
    |   movel([0.003745, -1.436740, -2.533940, -0.741710, 1.570796, 1.574542],accel_mss,speed_ms,0,blend_radius_m)
    |   movel([0.004739, -1.435848, -2.534641, -0.741899, 1.570796, 1.575536],accel_mss,speed_ms,0,blend_radius_m)
    |   movel([0.005272, -1.435530, -2.534892, -0.741967, 1.570796, 1.576068],accel_mss,speed_ms,0,blend_radius_m)
    |   movel([0.006401, -1.435122, -2.535212, -0.742055, 1.570796, 1.577198],accel_mss,speed_ms,0,blend_radius_m)
    |   movel([0.007590, -1.434991, -2.535315, -0.742083, 1.570796, 1.578387],accel_mss,speed_ms,0,blend_radius_m)
    |   movel([0.008814, -1.435103, -2.535227, -0.742059, 1.570796, 1.579611],accel_mss,speed_ms,0,blend_radius_m)
    |   movel([0.010051, -1.435426, -2.534974, -0.741990, 1.570796, 1.580848],accel_mss,speed_ms,0,blend_radius_m)
    |   movel([0.011275, -1.435920, -2.534585, -0.741884, 1.570796, 1.582071],accel_mss,speed_ms,0,blend_radius_m)
    |   movel([0.012464, -1.436554, -2.534086, -0.741749, 1.570796, 1.583260],accel_mss,speed_ms,0,blend_radius_m)
    |   movel([0.014637, -1.438088, -2.532876, -0.741425, 1.570796, 1.585434],accel_mss,speed_ms,0,blend_radius_m)
    |   movel([0.016390, -1.439747, -2.531563, -0.741079, 1.570796, 1.587186],accel_mss,speed_ms,0,blend_radius_m)
    |   movel([0.017549, -1.441238, -2.530380, -0.740771, 1.570796, 1.588345],accel_mss,speed_ms,0,blend_radius_m)
    |   movel([0.018583, -1.443176, -2.528837, -0.740376, 1.570796, 1.589380],accel_mss,speed_ms,0,blend_radius_m)
    |   movel([0.019434, -1.445226, -2.527199, -0.739965, 1.570796, 1.590230],accel_mss,speed_ms,0,blend_radius_m)
    |   movel([0.020761, -1.449528, -2.523739, -0.739122, 1.570796, 1.591558],accel_mss,speed_ms,0,blend_radius_m)
    |   movel([0.021881, -1.453903, -2.520192, -0.738294, 1.570796, 1.592678],accel_mss,speed_ms,0,blend_radius_m)
    |   movel([0.023134, -1.458118, -2.516746, -0.737525, 1.570796, 1.593931],accel_mss,speed_ms,0,blend_radius_m)
    |   movel([0.024538, -1.461727, -2.513775, -0.736888, 1.570796, 1.595335],accel_mss,speed_ms,0,blend_radius_m)
    |   movel([0.025445, -1.463393, -2.512395, -0.736601, 1.570796, 1.596242],accel_mss,speed_ms,0,blend_radius_m)
    |   movel([0.026600, -1.464881, -2.511160, -0.736348, 1.570796, 1.597396],accel_mss,speed_ms,0,blend_radius_m)
    |   movel([0.027285, -1.465459, -2.510679, -0.736250, 1.570796, 1.598081],accel_mss,speed_ms,0,blend_radius_m)
    |   movel([0.027711, -1.465654, -2.510517, -0.736218, 1.570796, 1.598507],accel_mss,speed_ms,0,blend_radius_m)
    |   movel([0.028210, -1.465744, -2.510442, -0.736203, 1.570796, 1.599006],accel_mss,speed_ms,0,blend_radius_m)
    |   movel([0.028929, -1.465671, -2.510503, -0.736215, 1.570796, 1.599725],accel_mss,speed_ms,0,blend_radius_m)
    |   movel([0.029678, -1.465424, -2.510708, -0.736256, 1.570796, 1.600475],accel_mss,speed_ms,0,blend_radius_m)
    |   movel([0.031166, -1.464617, -2.511380, -0.736392, 1.570796, 1.601962],accel_mss,speed_ms,0,blend_radius_m)
    |   movel([0.032779, -1.463512, -2.512297, -0.736580, 1.570796, 1.603576],accel_mss,speed_ms,0,blend_radius_m)
    |   movel([0.034310, -1.462320, -2.513284, -0.736785, 1.570796, 1.605106],accel_mss,speed_ms,0,blend_radius_m)
    |   movel([0.037186, -1.459741, -2.515412, -0.737236, 1.570796, 1.607982],accel_mss,speed_ms,0,blend_radius_m)
    |   movel([0.042702, -1.454304, -2.519865, -0.738220, 1.570796, 1.613498],accel_mss,speed_ms,0,blend_radius_m)
    |   movel([0.045403, -1.451829, -2.521877, -0.738683, 1.570796, 1.616199],accel_mss,speed_ms,0,blend_radius_m)
    |   movel([0.046992, -1.450531, -2.522928, -0.738930, 1.570796, 1.617788],accel_mss,speed_ms,0,blend_radius_m)
    |   movel([0.048604, -1.449412, -2.523833, -0.739144, 1.570796, 1.619400],accel_mss,speed_ms,0,blend_radius_m)
    |   movel([0.049387, -1.448969, -2.524190, -0.739230, 1.570796, 1.620183],accel_mss,speed_ms,0,blend_radius_m)
    |   movel([0.050139, -1.448633, -2.524461, -0.739295, 1.570796, 1.620936],accel_mss,speed_ms,0,blend_radius_m)
    |   movel([0.050846, -1.448423, -2.524631, -0.739336, 1.570796, 1.621642],accel_mss,speed_ms,0,blend_radius_m)
    |   movel([0.051495, -1.448361, -2.524681, -0.739348, 1.570796, 1.622291],accel_mss,speed_ms,0,blend_radius_m)
    |   movel([0.052072, -1.448464, -2.524597, -0.739328, 1.570796, 1.622869],accel_mss,speed_ms,0,blend_radius_m)
    |   movel([0.052567, -1.448754, -2.524364, -0.739271, 1.570796, 1.623363],accel_mss,speed_ms,0,blend_radius_m)
    |   movel([0.052966, -1.449251, -2.523962, -0.739175, 1.570796, 1.623763],accel_mss,speed_ms,0,blend_radius_m)
    |   movel([0.053255, -1.449976, -2.523377, -0.739036, 1.570796, 1.624051],accel_mss,speed_ms,0,blend_radius_m)
    |   movel([0.053543, -1.451361, -2.522257, -0.738772, 1.570796, 1.624340],accel_mss,speed_ms,0,blend_radius_m)
    |   movel([0.053666, -1.452775, -2.521109, -0.738505, 1.570796, 1.624462],accel_mss,speed_ms,0,blend_radius_m)
    |   movel([0.053632, -1.454212, -2.519940, -0.738237, 1.570796, 1.624429],accel_mss,speed_ms,0,blend_radius_m)
    |   movel([0.053453, -1.455671, -2.518750, -0.737968, 1.570796, 1.624249],accel_mss,speed_ms,0,blend_radius_m)
    |   movel([0.053133, -1.457143, -2.517546, -0.737700, 1.570796, 1.623929],accel_mss,speed_ms,0,blend_radius_m)
    |   movel([0.052683, -1.458624, -2.516331, -0.737434, 1.570796, 1.623479],accel_mss,speed_ms,0,blend_radius_m)
    |   movel([0.052110, -1.460111, -2.515108, -0.737171, 1.570796, 1.622906],accel_mss,speed_ms,0,blend_radius_m)
    |   movel([0.051424, -1.461599, -2.513880, -0.736910, 1.570796, 1.622220],accel_mss,speed_ms,0,blend_radius_m)
    |   movel([0.049747, -1.464556, -2.511430, -0.736403, 1.570796, 1.620543],accel_mss,speed_ms,0,blend_radius_m)
    |   movel([0.047714, -1.467466, -2.509006, -0.735917, 1.570796, 1.618510],accel_mss,speed_ms,0,blend_radius_m)
    |   movel([0.045389, -1.470294, -2.506638, -0.735457, 1.570796, 1.616185],accel_mss,speed_ms,0,blend_radius_m)
    |   movel([0.042838, -1.473006, -2.504355, -0.735028, 1.570796, 1.613634],accel_mss,speed_ms,0,blend_radius_m)
    |   movel([0.036899, -1.478881, -2.499370, -0.734138, 1.570796, 1.607695],accel_mss,speed_ms,0,blend_radius_m)
    |   movel([0.033733, -1.481692, -2.496966, -0.733731, 1.570796, 1.604529],accel_mss,speed_ms,0,blend_radius_m)
    |   movel([0.032106, -1.482978, -2.495862, -0.733549, 1.570796, 1.602902],accel_mss,speed_ms,0,blend_radius_m)
    |   movel([0.030449, -1.484152, -2.494851, -0.733385, 1.570796, 1.601246],accel_mss,speed_ms,0,blend_radius_m)
    |   movel([0.029367, -1.484827, -2.494270, -0.733292, 1.570796, 1.600163],accel_mss,speed_ms,0,blend_radius_m)
    |   movel([0.028277, -1.485408, -2.493769, -0.733212, 1.570796, 1.599074],accel_mss,speed_ms,0,blend_radius_m)
    |   movel([0.027188, -1.485882, -2.493359, -0.733148, 1.570796, 1.597984],accel_mss,speed_ms,0,blend_radius_m)
    |   movel([0.026108, -1.486237, -2.493053, -0.733100, 1.570796, 1.596904],accel_mss,speed_ms,0,blend_radius_m)
    |   movel([0.025048, -1.486460, -2.492860, -0.733070, 1.570796, 1.595844],accel_mss,speed_ms,0,blend_radius_m)
    |   movel([0.024014, -1.486539, -2.492791, -0.733059, 1.570796, 1.594811],accel_mss,speed_ms,0,blend_radius_m)
    |   movel([0.023018, -1.486457, -2.492862, -0.733070, 1.570796, 1.593814],accel_mss,speed_ms,0,blend_radius_m)
    |   movel([0.022065, -1.486202, -2.493082, -0.733104, 1.570796, 1.592861],accel_mss,speed_ms,0,blend_radius_m)
    |   movel([0.021200, -1.485770, -2.493456, -0.733163, 1.570796, 1.591996],accel_mss,speed_ms,0,blend_radius_m)
    |   movel([0.020477, -1.485214, -2.493936, -0.733239, 1.570796, 1.591274],accel_mss,speed_ms,0,blend_radius_m)
    |   movel([0.018046, -1.482555, -2.496225, -0.733609, 1.570796, 1.588843],accel_mss,speed_ms,0,blend_radius_m)
    |   movel([0.017307, -1.481986, -2.496714, -0.733689, 1.570796, 1.588104],accel_mss,speed_ms,0,blend_radius_m)
    |   movel([0.016416, -1.481539, -2.497097, -0.733753, 1.570796, 1.587212],accel_mss,speed_ms,0,blend_radius_m)
    |   movel([0.016011, -1.481473, -2.497154, -0.733762, 1.570796, 1.586808],accel_mss,speed_ms,0,blend_radius_m)
    |   movel([0.015826, -1.481649, -2.497003, -0.733737, 1.570796, 1.586622],accel_mss,speed_ms,0,blend_radius_m)
    |   movel([0.015586, -1.482106, -2.496611, -0.733672, 1.570796, 1.586383],accel_mss,speed_ms,0,blend_radius_m)
    |   movel([0.014967, -1.483715, -2.495228, -0.733446, 1.570796, 1.585763],accel_mss,speed_ms,0,blend_radius_m)
    |   movel([0.013426, -1.488626, -2.490982, -0.732781, 1.570796, 1.584223],accel_mss,speed_ms,0,blend_radius_m)
    |   movel([0.011008, -1.496849, -2.483788, -0.731753, 1.570796, 1.581805],accel_mss,speed_ms,0,blend_radius_m)
    |   movel([0.009222, -1.501167, -2.479967, -0.731255, 1.570796, 1.580018],accel_mss,speed_ms,0,blend_radius_m)
    |   movel([0.007219, -1.505451, -2.476146, -0.730791, 1.570796, 1.578016],accel_mss,speed_ms,0,blend_radius_m)
    |   movel([0.005025, -1.509696, -2.472332, -0.730360, 1.570796, 1.575822],accel_mss,speed_ms,0,blend_radius_m)
    |   movel([0.002672, -1.513892, -2.468534, -0.729963, 1.570796, 1.573469],accel_mss,speed_ms,0,blend_radius_m)
    |   movel([-0.000478, -1.519211, -2.463679, -0.729499, 1.570796, 1.570319],accel_mss,speed_ms,0,blend_radius_m)
    |   movel([-0.003754, -1.524489, -2.458816, -0.729083, 1.570796, 1.567042],accel_mss,speed_ms,0,blend_radius_m)
    |   movel([-0.007182, -1.529699, -2.453973, -0.728717, 1.570796, 1.563614],accel_mss,speed_ms,0,blend_radius_m)
    |   movel([-0.010795, -1.534808, -2.449181, -0.728400, 1.570796, 1.560002],accel_mss,speed_ms,0,blend_radius_m)
    |   movel([-0.014617, -1.539786, -2.444472, -0.728131, 1.570796, 1.556179],accel_mss,speed_ms,0,blend_radius_m)
    |   movel([-0.016614, -1.542217, -2.442157, -0.728015, 1.570796, 1.554182],accel_mss,speed_ms,0,blend_radius_m)
    |   movel([-0.018676, -1.544606, -2.439874, -0.727909, 1.570796, 1.552120],accel_mss,speed_ms,0,blend_radius_m)
    |   movel([-0.020806, -1.546949, -2.437625, -0.727815, 1.570796, 1.549991],accel_mss,speed_ms,0,blend_radius_m)
    |   movel([-0.023005, -1.549240, -2.435418, -0.727731, 1.570796, 1.547792],accel_mss,speed_ms,0,blend_radius_m)
    |   movel([-0.025277, -1.551481, -2.433251, -0.727657, 1.570796, 1.545519],accel_mss,speed_ms,0,blend_radius_m)
    |   movel([-0.027630, -1.553663, -2.431133, -0.727593, 1.570796, 1.543167],accel_mss,speed_ms,0,blend_radius_m)
    |   movel([-0.030515, -1.556180, -2.428680, -0.727529, 1.570796, 1.540281],accel_mss,speed_ms,0,blend_radius_m)
    |   movel([-0.032020, -1.557367, -2.427521, -0.727502, 1.570796, 1.538776],accel_mss,speed_ms,0,blend_radius_m)
    |   movel([-0.034729, -1.559211, -2.425714, -0.727465, 1.570796, 1.536067],accel_mss,speed_ms,0,blend_radius_m)
    |   movel([-0.036131, -1.560015, -2.424924, -0.727450, 1.570796, 1.534665],accel_mss,speed_ms,0,blend_radius_m)
    |   movel([-0.037535, -1.560590, -2.424358, -0.727440, 1.570796, 1.533261],accel_mss,speed_ms,0,blend_radius_m)
    |   movel([-0.038157, -1.560699, -2.424252, -0.727438, 1.570796, 1.532640],accel_mss,speed_ms,0,blend_radius_m)
    |   movel([-0.038686, -1.560641, -2.424308, -0.727439, 1.570796, 1.532111],accel_mss,speed_ms,0,blend_radius_m)
    |   movel([-0.038269, -1.559366, -2.425562, -0.727462, 1.570796, 1.532527],accel_mss,speed_ms,0,blend_radius_m)
    |   movel([-0.038057, -1.558114, -2.426789, -0.727486, 1.570796, 1.532739],accel_mss,speed_ms,0,blend_radius_m)
    |   movel([-0.038080, -1.557546, -2.427345, -0.727498, 1.570796, 1.532717],accel_mss,speed_ms,0,blend_radius_m)
    |   movel([-0.038217, -1.557042, -2.427838, -0.727509, 1.570796, 1.532579],accel_mss,speed_ms,0,blend_radius_m)
    |   movel([-0.038489, -1.556621, -2.428249, -0.727518, 1.570796, 1.532307],accel_mss,speed_ms,0,blend_radius_m)
    |   movel([-0.038922, -1.556307, -2.428557, -0.727526, 1.570796, 1.531874],accel_mss,speed_ms,0,blend_radius_m)
    |   movel([-0.040266, -1.555847, -2.429006, -0.727536, 1.570796, 1.530530],accel_mss,speed_ms,0,blend_radius_m)
    |   movel([-0.040634, -1.555571, -2.429275, -0.727543, 1.570796, 1.530162],accel_mss,speed_ms,0,blend_radius_m)
    |   movel([-0.040882, -1.555212, -2.429625, -0.727552, 1.570796, 1.529914],accel_mss,speed_ms,0,blend_radius_m)
    |   movel([-0.041069, -1.554306, -2.430507, -0.727576, 1.570796, 1.529727],accel_mss,speed_ms,0,blend_radius_m)
    |   movel([-0.040955, -1.553246, -2.431538, -0.727605, 1.570796, 1.529841],accel_mss,speed_ms,0,blend_radius_m)
    |   movel([-0.040664, -1.552156, -2.432596, -0.727636, 1.570796, 1.530133],accel_mss,speed_ms,0,blend_radius_m)
    |   movel([-0.039553, -1.548866, -2.435779, -0.727744, 1.570796, 1.531243],accel_mss,speed_ms,0,blend_radius_m)
    |   movel([-0.038218, -1.545533, -2.438985, -0.727871, 1.570796, 1.532578],accel_mss,speed_ms,0,blend_radius_m)
    |   movel([-0.037429, -1.543870, -2.440578, -0.727941, 1.570796, 1.533368],accel_mss,speed_ms,0,blend_radius_m)
    |   movel([-0.036541, -1.542216, -2.442158, -0.728015, 1.570796, 1.534255],accel_mss,speed_ms,0,blend_radius_m)
    |   movel([-0.035539, -1.540583, -2.443714, -0.728092, 1.570796, 1.535257],accel_mss,speed_ms,0,blend_radius_m)
    |   movel([-0.034409, -1.538975, -2.445242, -0.728172, 1.570796, 1.536388],accel_mss,speed_ms,0,blend_radius_m)
    |   movel([-0.033134, -1.537476, -2.446662, -0.728251, 1.570796, 1.537662],accel_mss,speed_ms,0,blend_radius_m)
    |   movel([-0.028906, -1.533326, -2.450576, -0.728488, 1.570796, 1.541890],accel_mss,speed_ms,0,blend_radius_m)
    |   movel([-0.025637, -1.529653, -2.454016, -0.728720, 1.570796, 1.545159],accel_mss,speed_ms,0,blend_radius_m)
    |   movel([-0.022466, -1.525894, -2.457515, -0.728980, 1.570796, 1.548330],accel_mss,speed_ms,0,blend_radius_m)
    |   movel([-0.021068, -1.524181, -2.459101, -0.729106, 1.570796, 1.549729],accel_mss,speed_ms,0,blend_radius_m)
    |   speed_ms = 0.005
    |   movel([-0.021068, -1.516515, -2.455705, -0.740169, 1.570796, 1.549729],accel_mss,speed_ms,0,blend_radius_m)
    |   speed_ms = 0.040
    |   movel([-0.050485, -1.547182, -2.426938, -0.738269, 1.570796, 1.520312],accel_mss,speed_ms,0,blend_radius_m)
    |   speed_ms = 0.005
    |   movel([-0.050485, -1.554601, -2.430220, -0.727568, 1.570796, 1.520312],accel_mss,speed_ms,0,blend_radius_m)
    |   speed_ms = 0.025
    |   movel([-0.048077, -1.556856, -2.428020, -0.727513, 1.570796, 1.522719],accel_mss,speed_ms,0,blend_radius_m)
    |   movel([-0.046893, -1.558135, -2.426768, -0.727486, 1.570796, 1.523903],accel_mss,speed_ms,0,blend_radius_m)
    |   movel([-0.045817, -1.559516, -2.425414, -0.727459, 1.570796, 1.524979],accel_mss,speed_ms,0,blend_radius_m)
    |   movel([-0.044913, -1.560988, -2.423967, -0.727434, 1.570796, 1.525883],accel_mss,speed_ms,0,blend_radius_m)
    |   movel([-0.044250, -1.562548, -2.422429, -0.727411, 1.570796, 1.526546],accel_mss,speed_ms,0,blend_radius_m)
    |   movel([-0.043895, -1.564194, -2.420804, -0.727391, 1.570796, 1.526901],accel_mss,speed_ms,0,blend_radius_m)
    |   movel([-0.043854, -1.565048, -2.419958, -0.727383, 1.570796, 1.526942],accel_mss,speed_ms,0,blend_radius_m)
    |   movel([-0.043915, -1.565919, -2.419095, -0.727375, 1.570796, 1.526881],accel_mss,speed_ms,0,blend_radius_m)
    |   movel([-0.044514, -1.565604, -2.419407, -0.727378, 1.570796, 1.526282],accel_mss,speed_ms,0,blend_radius_m)
    |   movel([-0.044896, -1.565193, -2.419815, -0.727382, 1.570796, 1.525901],accel_mss,speed_ms,0,blend_radius_m)
    |   movel([-0.045696, -1.564234, -2.420764, -0.727391, 1.570796, 1.525100],accel_mss,speed_ms,0,blend_radius_m)
    |   movel([-0.046816, -1.563414, -2.421575, -0.727400, 1.570796, 1.523981],accel_mss,speed_ms,0,blend_radius_m)
    |   movel([-0.048058, -1.562711, -2.422269, -0.727409, 1.570796, 1.522738],accel_mss,speed_ms,0,blend_radius_m)
    |   movel([-0.049410, -1.562120, -2.422852, -0.727417, 1.570796, 1.521386],accel_mss,speed_ms,0,blend_radius_m)
    |   movel([-0.050857, -1.561642, -2.423323, -0.727424, 1.570796, 1.519939],accel_mss,speed_ms,0,blend_radius_m)
    |   movel([-0.052384, -1.561274, -2.423686, -0.727429, 1.570796, 1.518413],accel_mss,speed_ms,0,blend_radius_m)
    |   movel([-0.053976, -1.561017, -2.423938, -0.727433, 1.570796, 1.516821],accel_mss,speed_ms,0,blend_radius_m)
    |   movel([-0.055620, -1.560871, -2.424083, -0.727436, 1.570796, 1.515177],accel_mss,speed_ms,0,blend_radius_m)
    |   movel([-0.057299, -1.560831, -2.424122, -0.727436, 1.570796, 1.513497],accel_mss,speed_ms,0,blend_radius_m)
    |   movel([-0.058436, -1.560890, -2.424063, -0.727435, 1.570796, 1.512360],accel_mss,speed_ms,0,blend_radius_m)
    |   movel([-0.059341, -1.561045, -2.423911, -0.727433, 1.570796, 1.511456],accel_mss,speed_ms,0,blend_radius_m)
    |   movel([-0.060029, -1.561283, -2.423677, -0.727429, 1.570796, 1.510767],accel_mss,speed_ms,0,blend_radius_m)
    |   movel([-0.060522, -1.561594, -2.423370, -0.727425, 1.570796, 1.510275],accel_mss,speed_ms,0,blend_radius_m)
    |   movel([-0.060839, -1.561972, -2.422998, -0.727419, 1.570796, 1.509957],accel_mss,speed_ms,0,blend_radius_m)
    |   movel([-0.060998, -1.562406, -2.422570, -0.727413, 1.570796, 1.509798],accel_mss,speed_ms,0,blend_radius_m)
    |   movel([-0.061024, -1.562886, -2.422096, -0.727407, 1.570796, 1.509773],accel_mss,speed_ms,0,blend_radius_m)
    |   movel([-0.060930, -1.563404, -2.421585, -0.727400, 1.570796, 1.509866],accel_mss,speed_ms,0,blend_radius_m)
    |   movel([-0.060476, -1.564519, -2.420482, -0.727388, 1.570796, 1.510321],accel_mss,speed_ms,0,blend_radius_m)
    |   movel([-0.058367, -1.567859, -2.417166, -0.727363, 1.570796, 1.512429],accel_mss,speed_ms,0,blend_radius_m)
    |   movel([-0.059813, -1.566992, -2.418029, -0.727368, 1.570796, 1.510983],accel_mss,speed_ms,0,blend_radius_m)
    |   movel([-0.062636, -1.565198, -2.419810, -0.727382, 1.570796, 1.508160],accel_mss,speed_ms,0,blend_radius_m)
    |   movel([-0.064238, -1.564514, -2.420487, -0.727388, 1.570796, 1.506559],accel_mss,speed_ms,0,blend_radius_m)
    |   movel([-0.066175, -1.563972, -2.421023, -0.727394, 1.570796, 1.504621],accel_mss,speed_ms,0,blend_radius_m)
    |   movel([-0.068188, -1.563525, -2.421465, -0.727399, 1.570796, 1.502609],accel_mss,speed_ms,0,blend_radius_m)
    |   movel([-0.072264, -1.562702, -2.422278, -0.727409, 1.570796, 1.498533],accel_mss,speed_ms,0,blend_radius_m)
    |   movel([-0.074241, -1.562223, -2.422750, -0.727416, 1.570796, 1.496555],accel_mss,speed_ms,0,blend_radius_m)
    |   movel([-0.076119, -1.561629, -2.423336, -0.727424, 1.570796, 1.494677],accel_mss,speed_ms,0,blend_radius_m)
    |   movel([-0.077854, -1.560870, -2.424083, -0.727436, 1.570796, 1.492942],accel_mss,speed_ms,0,blend_radius_m)
    |   movel([-0.079405, -1.559889, -2.425047, -0.727452, 1.570796, 1.491391],accel_mss,speed_ms,0,blend_radius_m)
    |   movel([-0.078004, -1.562788, -2.422193, -0.727408, 1.570796, 1.492793],accel_mss,speed_ms,0,blend_radius_m)
    |   movel([-0.077190, -1.564223, -2.420774, -0.727391, 1.570796, 1.493606],accel_mss,speed_ms,0,blend_radius_m)
    |   movel([-0.076252, -1.565437, -2.419572, -0.727379, 1.570796, 1.494544],accel_mss,speed_ms,0,blend_radius_m)
    |   movel([-0.077828, -1.564527, -2.420474, -0.727388, 1.570796, 1.492968],accel_mss,speed_ms,0,blend_radius_m)
    |   movel([-0.079555, -1.563782, -2.421211, -0.727396, 1.570796, 1.491241],accel_mss,speed_ms,0,blend_radius_m)
    |   movel([-0.083157, -1.562454, -2.422523, -0.727412, 1.570796, 1.487639],accel_mss,speed_ms,0,blend_radius_m)
    |   movel([-0.084295, -1.561925, -2.423044, -0.727420, 1.570796, 1.486502],accel_mss,speed_ms,0,blend_radius_m)
    |   movel([-0.085304, -1.561305, -2.423655, -0.727429, 1.570796, 1.485493],accel_mss,speed_ms,0,blend_radius_m)
    |   movel([-0.087071, -1.559876, -2.425061, -0.727452, 1.570796, 1.483725],accel_mss,speed_ms,0,blend_radius_m)
    |   movel([-0.088743, -1.558350, -2.426558, -0.727481, 1.570796, 1.482053],accel_mss,speed_ms,0,blend_radius_m)
    |   movel([-0.090604, -1.556919, -2.427959, -0.727512, 1.570796, 1.480192],accel_mss,speed_ms,0,blend_radius_m)
    |   movel([-0.091273, -1.556544, -2.428325, -0.727520, 1.570796, 1.479524],accel_mss,speed_ms,0,blend_radius_m)
    |   movel([-0.092029, -1.556274, -2.428589, -0.727526, 1.570796, 1.478767],accel_mss,speed_ms,0,blend_radius_m)
    |   movel([-0.092868, -1.556196, -2.428664, -0.727528, 1.570796, 1.477929],accel_mss,speed_ms,0,blend_radius_m)
    |   movel([-0.093312, -1.556253, -2.428609, -0.727527, 1.570796, 1.477485],accel_mss,speed_ms,0,blend_radius_m)
    |   movel([-0.093773, -1.556392, -2.428473, -0.727524, 1.570796, 1.477023],accel_mss,speed_ms,0,blend_radius_m)
    |   movel([-0.094268, -1.556630, -2.428241, -0.727518, 1.570796, 1.476529],accel_mss,speed_ms,0,blend_radius_m)
    |   movel([-0.094711, -1.556935, -2.427942, -0.727511, 1.570796, 1.476085],accel_mss,speed_ms,0,blend_radius_m)
    |   movel([-0.095469, -1.557702, -2.427192, -0.727495, 1.570796, 1.475328],accel_mss,speed_ms,0,blend_radius_m)
    |   movel([-0.096070, -1.558593, -2.426319, -0.727476, 1.570796, 1.474726],accel_mss,speed_ms,0,blend_radius_m)
    |   movel([-0.096540, -1.559509, -2.425421, -0.727459, 1.570796, 1.474256],accel_mss,speed_ms,0,blend_radius_m)
    |   movel([-0.097023, -1.558082, -2.426821, -0.727487, 1.570796, 1.473773],accel_mss,speed_ms,0,blend_radius_m)
    |   movel([-0.097641, -1.556752, -2.428121, -0.727515, 1.570796, 1.473155],accel_mss,speed_ms,0,blend_radius_m)
    |   movel([-0.099137, -1.554288, -2.430525, -0.727576, 1.570796, 1.471659],accel_mss,speed_ms,0,blend_radius_m)
    |   movel([-0.100733, -1.551892, -2.432852, -0.727644, 1.570796, 1.470064],accel_mss,speed_ms,0,blend_radius_m)
    |   movel([-0.102125, -1.549338, -2.435323, -0.727727, 1.570796, 1.468671],accel_mss,speed_ms,0,blend_radius_m)
    |   movel([-0.102491, -1.548250, -2.436373, -0.727766, 1.570796, 1.468306],accel_mss,speed_ms,0,blend_radius_m)
    |   movel([-0.102692, -1.547057, -2.437521, -0.727811, 1.570796, 1.468104],accel_mss,speed_ms,0,blend_radius_m)
    |   movel([-0.102755, -1.545783, -2.438746, -0.727861, 1.570796, 1.468042],accel_mss,speed_ms,0,blend_radius_m)
    |   movel([-0.102703, -1.544455, -2.440019, -0.727916, 1.570796, 1.468094],accel_mss,speed_ms,0,blend_radius_m)
    |   movel([-0.102341, -1.541729, -2.442622, -0.728037, 1.570796, 1.468456],accel_mss,speed_ms,0,blend_radius_m)
    |   movel([-0.101797, -1.539085, -2.445137, -0.728167, 1.570796, 1.468999],accel_mss,speed_ms,0,blend_radius_m)
    |   speed_ms = 0.005
    |   movel([-0.101797, -1.531540, -2.441797, -0.739052, 1.570796, 1.468999],accel_mss,speed_ms,0,blend_radius_m)
    |   speed_ms = 0.040
    |   # Splitting Linear movement in 2 (instruction 806: MoveL 765)
    |   movel([-0.083040, -1.496373, -2.473790, -0.742226, 1.570796, 1.487756],accel_mss,speed_ms,0,blend_radius_m)
    |   movel([-0.062711, -1.459410, -2.505329, -0.747649, 1.570796, 1.508085],accel_mss,speed_ms,0,blend_radius_m)
    |   speed_ms = 0.005
    |   movel([-0.062711, -1.467532, -2.508951, -0.735906, 1.570796, 1.508085],accel_mss,speed_ms,0,blend_radius_m)
    |   speed_ms = 0.025
    |   movel([-0.063837, -1.468399, -2.508227, -0.735764, 1.570796, 1.506960],accel_mss,speed_ms,0,blend_radius_m)
    |   movel([-0.063923, -1.468577, -2.508077, -0.735735, 1.570796, 1.506874],accel_mss,speed_ms,0,blend_radius_m)
    |   movel([-0.063841, -1.468838, -2.507859, -0.735692, 1.570796, 1.506955],accel_mss,speed_ms,0,blend_radius_m)
    |   movel([-0.063219, -1.469593, -2.507226, -0.735570, 1.570796, 1.507577],accel_mss,speed_ms,0,blend_radius_m)
    |   movel([-0.060441, -1.471875, -2.505309, -0.735205, 1.570796, 1.510355],accel_mss,speed_ms,0,blend_radius_m)
    |   movel([-0.056183, -1.474894, -2.502759, -0.734736, 1.570796, 1.514613],accel_mss,speed_ms,0,blend_radius_m)
    |   movel([-0.051114, -1.478295, -2.499870, -0.734224, 1.570796, 1.519682],accel_mss,speed_ms,0,blend_radius_m)
    |   movel([-0.041146, -1.484794, -2.494299, -0.733297, 1.570796, 1.529651],accel_mss,speed_ms,0,blend_radius_m)
    |   movel([-0.035496, -1.488354, -2.491218, -0.732817, 1.570796, 1.535301],accel_mss,speed_ms,0,blend_radius_m)
    |   movel([-0.034943, -1.488610, -2.490996, -0.732783, 1.570796, 1.535853],accel_mss,speed_ms,0,blend_radius_m)
    |   movel([-0.034315, -1.488765, -2.490861, -0.732763, 1.570796, 1.536482],accel_mss,speed_ms,0,blend_radius_m)
    |   movel([-0.033650, -1.488731, -2.490891, -0.732767, 1.570796, 1.537147],accel_mss,speed_ms,0,blend_radius_m)
    |   movel([-0.033313, -1.488618, -2.490989, -0.732782, 1.570796, 1.537483],accel_mss,speed_ms,0,blend_radius_m)
    |   movel([-0.032983, -1.488424, -2.491157, -0.732807, 1.570796, 1.537814],accel_mss,speed_ms,0,blend_radius_m)
    |   movel([-0.032497, -1.487936, -2.491581, -0.732872, 1.570796, 1.538299],accel_mss,speed_ms,0,blend_radius_m)
    |   movel([-0.032145, -1.487377, -2.492066, -0.732946, 1.570796, 1.538651],accel_mss,speed_ms,0,blend_radius_m)
    |   movel([-0.030514, -1.484185, -2.494823, -0.733381, 1.570796, 1.540282],accel_mss,speed_ms,0,blend_radius_m)
    |   movel([-0.029155, -1.480964, -2.497589, -0.733835, 1.570796, 1.541641],accel_mss,speed_ms,0,blend_radius_m)
    |   movel([-0.028056, -1.477733, -2.500349, -0.734307, 1.570796, 1.542740],accel_mss,speed_ms,0,blend_radius_m)
    |   movel([-0.027194, -1.474507, -2.503087, -0.734795, 1.570796, 1.543603],accel_mss,speed_ms,0,blend_radius_m)
    |   movel([-0.026554, -1.471302, -2.505791, -0.735296, 1.570796, 1.544242],accel_mss,speed_ms,0,blend_radius_m)
    |   movel([-0.026117, -1.468135, -2.508447, -0.735807, 1.570796, 1.544679],accel_mss,speed_ms,0,blend_radius_m)
    |   movel([-0.025866, -1.465023, -2.511042, -0.736324, 1.570796, 1.544931],accel_mss,speed_ms,0,blend_radius_m)
    |   movel([-0.025780, -1.461986, -2.513560, -0.736843, 1.570796, 1.545016],accel_mss,speed_ms,0,blend_radius_m)
    |   movel([-0.025847, -1.460637, -2.514674, -0.737078, 1.570796, 1.544950],accel_mss,speed_ms,0,blend_radius_m)
    |   movel([-0.026050, -1.459421, -2.515675, -0.737292, 1.570796, 1.544746],accel_mss,speed_ms,0,blend_radius_m)
    |   movel([-0.026390, -1.458337, -2.516566, -0.737486, 1.570796, 1.544407],accel_mss,speed_ms,0,blend_radius_m)
    |   movel([-0.026856, -1.457380, -2.517351, -0.737657, 1.570796, 1.543941],accel_mss,speed_ms,0,blend_radius_m)
    |   movel([-0.027447, -1.456551, -2.518030, -0.737808, 1.570796, 1.543349],accel_mss,speed_ms,0,blend_radius_m)
    |   movel([-0.028158, -1.455848, -2.518605, -0.737936, 1.570796, 1.542638],accel_mss,speed_ms,0,blend_radius_m)
    |   movel([-0.028984, -1.455264, -2.519082, -0.738043, 1.570796, 1.541812],accel_mss,speed_ms,0,blend_radius_m)
    |   movel([-0.029921, -1.454799, -2.519462, -0.738128, 1.570796, 1.540875],accel_mss,speed_ms,0,blend_radius_m)
    |   movel([-0.030963, -1.454450, -2.519746, -0.738193, 1.570796, 1.539834],accel_mss,speed_ms,0,blend_radius_m)
    |   movel([-0.032104, -1.454214, -2.519938, -0.738236, 1.570796, 1.538692],accel_mss,speed_ms,0,blend_radius_m)
    |   movel([-0.033343, -1.454088, -2.520041, -0.738260, 1.570796, 1.537453],accel_mss,speed_ms,0,blend_radius_m)
    |   movel([-0.034670, -1.454070, -2.520056, -0.738263, 1.570796, 1.536126],accel_mss,speed_ms,0,blend_radius_m)
    |   movel([-0.037577, -1.454345, -2.519832, -0.738212, 1.570796, 1.533220],accel_mss,speed_ms,0,blend_radius_m)
    |   movel([-0.040780, -1.455010, -2.519289, -0.738089, 1.570796, 1.530016],accel_mss,speed_ms,0,blend_radius_m)
    |   movel([-0.043678, -1.455908, -2.518556, -0.737925, 1.570796, 1.527118],accel_mss,speed_ms,0,blend_radius_m)
    |   movel([-0.046535, -1.457075, -2.517601, -0.737713, 1.570796, 1.524261],accel_mss,speed_ms,0,blend_radius_m)
    |   movel([-0.049352, -1.458477, -2.516452, -0.737461, 1.570796, 1.521445],accel_mss,speed_ms,0,blend_radius_m)
    |   movel([-0.052124, -1.460068, -2.515143, -0.737178, 1.570796, 1.518673],accel_mss,speed_ms,0,blend_radius_m)
    |   movel([-0.054845, -1.461809, -2.513706, -0.736874, 1.570796, 1.515951],accel_mss,speed_ms,0,blend_radius_m)
    |   movel([-0.057519, -1.463659, -2.512174, -0.736555, 1.570796, 1.513277],accel_mss,speed_ms,0,blend_radius_m)
    |   movel([-0.062711, -1.467532, -2.508951, -0.735906, 1.570796, 1.508085],accel_mss,speed_ms,0,blend_radius_m)
    |   movel([-0.063837, -1.468399, -2.508227, -0.735764, 1.570796, 1.506960],accel_mss,speed_ms,0,blend_radius_m)
    |   movel([-0.063923, -1.468577, -2.508077, -0.735735, 1.570796, 1.506874],accel_mss,speed_ms,0,blend_radius_m)
    |   movel([-0.063841, -1.468838, -2.507859, -0.735692, 1.570796, 1.506955],accel_mss,speed_ms,0,blend_radius_m)
    |   movel([-0.063645, -1.469078, -2.507658, -0.735653, 1.570796, 1.507152],accel_mss,speed_ms,0,blend_radius_m)
    |   speed_ms = 0.005
    |   movel([-0.063645, -1.460968, -2.504043, -0.747378, 1.570796, 1.507152],accel_mss,speed_ms,0,blend_radius_m)
    |   speed_ms = 0.040
    |   movel([-0.072174, -1.446258, -2.516044, -0.750087, 1.570796, 1.498622],accel_mss,speed_ms,0,blend_radius_m)
    |   speed_ms = 0.005
    |   movel([-0.072174, -1.454482, -2.519720, -0.738187, 1.570796, 1.498622],accel_mss,speed_ms,0,blend_radius_m)
    |   speed_ms = 0.025
    |   movel([-0.072243, -1.453237, -2.520734, -0.738418, 1.570796, 1.498554],accel_mss,speed_ms,0,blend_radius_m)
    |   movel([-0.072544, -1.452088, -2.521667, -0.738634, 1.570796, 1.498253],accel_mss,speed_ms,0,blend_radius_m)
    |   movel([-0.073071, -1.451063, -2.522498, -0.738828, 1.570796, 1.497725],accel_mss,speed_ms,0,blend_radius_m)
    |   movel([-0.073812, -1.450185, -2.523208, -0.738996, 1.570796, 1.496985],accel_mss,speed_ms,0,blend_radius_m)
    |   movel([-0.076104, -1.448426, -2.524628, -0.739335, 1.570796, 1.494692],accel_mss,speed_ms,0,blend_radius_m)
    |   movel([-0.076657, -1.447844, -2.525096, -0.739448, 1.570796, 1.494140],accel_mss,speed_ms,0,blend_radius_m)
    |   movel([-0.077038, -1.447218, -2.525600, -0.739571, 1.570796, 1.493758],accel_mss,speed_ms,0,blend_radius_m)
    |   movel([-0.077170, -1.446555, -2.526133, -0.739701, 1.570796, 1.493626],accel_mss,speed_ms,0,blend_radius_m)
    |   movel([-0.076970, -1.445860, -2.526690, -0.739838, 1.570796, 1.493826],accel_mss,speed_ms,0,blend_radius_m)
    |   movel([-0.076391, -1.445103, -2.527297, -0.739989, 1.570796, 1.494405],accel_mss,speed_ms,0,blend_radius_m)
    |   movel([-0.075691, -1.444616, -2.527687, -0.740086, 1.570796, 1.495105],accel_mss,speed_ms,0,blend_radius_m)
    |   movel([-0.074908, -1.444355, -2.527895, -0.740138, 1.570796, 1.495888],accel_mss,speed_ms,0,blend_radius_m)
    |   movel([-0.074087, -1.444277, -2.527958, -0.740154, 1.570796, 1.496710],accel_mss,speed_ms,0,blend_radius_m)
    |   movel([-0.072504, -1.444494, -2.527784, -0.740111, 1.570796, 1.498293],accel_mss,speed_ms,0,blend_radius_m)
    |   movel([-0.071273, -1.444919, -2.527445, -0.740026, 1.570796, 1.499523],accel_mss,speed_ms,0,blend_radius_m)
    |   movel([-0.071721, -1.443489, -2.528587, -0.740313, 1.570796, 1.499075],accel_mss,speed_ms,0,blend_radius_m)
    |   movel([-0.072443, -1.442254, -2.529572, -0.740563, 1.570796, 1.498354],accel_mss,speed_ms,0,blend_radius_m)
    |   movel([-0.074382, -1.440116, -2.531271, -0.741002, 1.570796, 1.496414],accel_mss,speed_ms,0,blend_radius_m)
    |   movel([-0.076427, -1.437995, -2.532949, -0.741445, 1.570796, 1.494369],accel_mss,speed_ms,0,blend_radius_m)
    |   movel([-0.077282, -1.436778, -2.533909, -0.741702, 1.570796, 1.493514],accel_mss,speed_ms,0,blend_radius_m)
    |   movel([-0.077910, -1.435370, -2.535018, -0.742002, 1.570796, 1.492887],accel_mss,speed_ms,0,blend_radius_m)
    |   movel([-0.078155, -1.434398, -2.535780, -0.742211, 1.570796, 1.492641],accel_mss,speed_ms,0,blend_radius_m)
    |   movel([-0.078235, -1.433559, -2.536438, -0.742392, 1.570796, 1.492561],accel_mss,speed_ms,0,blend_radius_m)
    |   movel([-0.078168, -1.432849, -2.536994, -0.742547, 1.570796, 1.492628],accel_mss,speed_ms,0,blend_radius_m)
    |   movel([-0.077968, -1.432265, -2.537450, -0.742674, 1.570796, 1.492829],accel_mss,speed_ms,0,blend_radius_m)
    |   movel([-0.077656, -1.431807, -2.537808, -0.742775, 1.570796, 1.493140],accel_mss,speed_ms,0,blend_radius_m)
    |   movel([-0.077247, -1.431464, -2.538075, -0.742850, 1.570796, 1.493549],accel_mss,speed_ms,0,blend_radius_m)
    |   movel([-0.076762, -1.431238, -2.538251, -0.742900, 1.570796, 1.494034],accel_mss,speed_ms,0,blend_radius_m)
    |   movel([-0.076215, -1.431124, -2.538340, -0.742925, 1.570796, 1.494581],accel_mss,speed_ms,0,blend_radius_m)
    |   movel([-0.075625, -1.431117, -2.538345, -0.742926, 1.570796, 1.495171],accel_mss,speed_ms,0,blend_radius_m)
    |   movel([-0.075014, -1.431216, -2.538268, -0.742905, 1.570796, 1.495783],accel_mss,speed_ms,0,blend_radius_m)
    |   movel([-0.073786, -1.431708, -2.537885, -0.742796, 1.570796, 1.497010],accel_mss,speed_ms,0,blend_radius_m)
    |   movel([-0.072674, -1.432567, -2.537214, -0.742608, 1.570796, 1.498122],accel_mss,speed_ms,0,blend_radius_m)
    |   movel([-0.071818, -1.433760, -2.536280, -0.742348, 1.570796, 1.498978],accel_mss,speed_ms,0,blend_radius_m)
    |   movel([-0.071570, -1.432334, -2.537396, -0.742659, 1.570796, 1.499226],accel_mss,speed_ms,0,blend_radius_m)
    |   movel([-0.071523, -1.431037, -2.538408, -0.742944, 1.570796, 1.499273],accel_mss,speed_ms,0,blend_radius_m)
    |   movel([-0.071633, -1.429838, -2.539341, -0.743210, 1.570796, 1.499163],accel_mss,speed_ms,0,blend_radius_m)
    |   movel([-0.072441, -1.426473, -2.541948, -0.743968, 1.570796, 1.498355],accel_mss,speed_ms,0,blend_radius_m)
    |   movel([-0.072913, -1.424072, -2.543798, -0.744519, 1.570796, 1.497883],accel_mss,speed_ms,0,blend_radius_m)
    |   movel([-0.072968, -1.423023, -2.544604, -0.744762, 1.570796, 1.497829],accel_mss,speed_ms,0,blend_radius_m)
    |   movel([-0.072889, -1.422073, -2.545332, -0.744984, 1.570796, 1.497908],accel_mss,speed_ms,0,blend_radius_m)
    |   movel([-0.072695, -1.421230, -2.545977, -0.745182, 1.570796, 1.498101],accel_mss,speed_ms,0,blend_radius_m)
    |   movel([-0.072401, -1.420498, -2.546536, -0.745355, 1.570796, 1.498395],accel_mss,speed_ms,0,blend_radius_m)
    |   movel([-0.072027, -1.419881, -2.547006, -0.745502, 1.570796, 1.498770],accel_mss,speed_ms,0,blend_radius_m)
    |   movel([-0.071586, -1.419384, -2.547385, -0.745620, 1.570796, 1.499210],accel_mss,speed_ms,0,blend_radius_m)
    |   movel([-0.071096, -1.419012, -2.547668, -0.745709, 1.570796, 1.499700],accel_mss,speed_ms,0,blend_radius_m)
    |   movel([-0.070575, -1.418770, -2.547852, -0.745766, 1.570796, 1.500221],accel_mss,speed_ms,0,blend_radius_m)
    |   movel([-0.070039, -1.418663, -2.547934, -0.745792, 1.570796, 1.500757],accel_mss,speed_ms,0,blend_radius_m)
    |   movel([-0.069506, -1.418695, -2.547909, -0.745784, 1.570796, 1.501291],accel_mss,speed_ms,0,blend_radius_m)
    |   movel([-0.068990, -1.418869, -2.547777, -0.745743, 1.570796, 1.501806],accel_mss,speed_ms,0,blend_radius_m)
    |   movel([-0.068509, -1.419192, -2.547531, -0.745666, 1.570796, 1.502287],accel_mss,speed_ms,0,blend_radius_m)
    |   movel([-0.068083, -1.419668, -2.547169, -0.745552, 1.570796, 1.502713],accel_mss,speed_ms,0,blend_radius_m)
    |   movel([-0.067726, -1.420299, -2.546687, -0.745402, 1.570796, 1.503070],accel_mss,speed_ms,0,blend_radius_m)
    |   movel([-0.067456, -1.421092, -2.546082, -0.745215, 1.570796, 1.503341],accel_mss,speed_ms,0,blend_radius_m)
    |   movel([-0.067286, -1.422046, -2.545352, -0.744991, 1.570796, 1.503511],accel_mss,speed_ms,0,blend_radius_m)
    |   movel([-0.066480, -1.420784, -2.546318, -0.745288, 1.570796, 1.504317],accel_mss,speed_ms,0,blend_radius_m)
    |   movel([-0.065836, -1.419517, -2.547284, -0.745588, 1.570796, 1.504961],accel_mss,speed_ms,0,blend_radius_m)
    |   movel([-0.065321, -1.418247, -2.548250, -0.745892, 1.570796, 1.505475],accel_mss,speed_ms,0,blend_radius_m)
    |   movel([-0.064903, -1.416973, -2.549217, -0.746199, 1.570796, 1.505893],accel_mss,speed_ms,0,blend_radius_m)
    |   movel([-0.063493, -1.411871, -2.553065, -0.747453, 1.570796, 1.507303],accel_mss,speed_ms,0,blend_radius_m)
    |   movel([-0.062918, -1.409984, -2.554478, -0.747927, 1.570796, 1.507878],accel_mss,speed_ms,0,blend_radius_m)
    |   movel([-0.062028, -1.407742, -2.556150, -0.748496, 1.570796, 1.508768],accel_mss,speed_ms,0,blend_radius_m)
    |   movel([-0.061398, -1.406679, -2.556941, -0.748769, 1.570796, 1.509398],accel_mss,speed_ms,0,blend_radius_m)
    |   movel([-0.060609, -1.405759, -2.557623, -0.749006, 1.570796, 1.510187],accel_mss,speed_ms,0,blend_radius_m)
    |   movel([-0.060144, -1.405377, -2.557906, -0.749106, 1.570796, 1.510652],accel_mss,speed_ms,0,blend_radius_m)
    |   movel([-0.059065, -1.404813, -2.558324, -0.749252, 1.570796, 1.511731],accel_mss,speed_ms,0,blend_radius_m)
    |   movel([-0.058441, -1.404655, -2.558441, -0.749293, 1.570796, 1.512355],accel_mss,speed_ms,0,blend_radius_m)
    |   movel([-0.057834, -1.404687, -2.558417, -0.749285, 1.570796, 1.512962],accel_mss,speed_ms,0,blend_radius_m)
    |   movel([-0.057396, -1.404971, -2.558207, -0.749211, 1.570796, 1.513400],accel_mss,speed_ms,0,blend_radius_m)
    |   movel([-0.056907, -1.405936, -2.557492, -0.748961, 1.570796, 1.513889],accel_mss,speed_ms,0,blend_radius_m)
    |   movel([-0.056592, -1.407441, -2.556375, -0.748574, 1.570796, 1.514204],accel_mss,speed_ms,0,blend_radius_m)
    |   movel([-0.056446, -1.409015, -2.555202, -0.748172, 1.570796, 1.514350],accel_mss,speed_ms,0,blend_radius_m)
    |   movel([-0.055172, -1.407309, -2.556473, -0.748607, 1.570796, 1.515625],accel_mss,speed_ms,0,blend_radius_m)
    |   movel([-0.053733, -1.405654, -2.557701, -0.749034, 1.570796, 1.517063],accel_mss,speed_ms,0,blend_radius_m)
    |   movel([-0.052159, -1.404070, -2.558873, -0.749446, 1.570796, 1.518637],accel_mss,speed_ms,0,blend_radius_m)
    |   movel([-0.050484, -1.402575, -2.559976, -0.749838, 1.570796, 1.520313],accel_mss,speed_ms,0,blend_radius_m)
    |   movel([-0.047138, -1.399585, -2.562172, -0.750632, 1.570796, 1.523659],accel_mss,speed_ms,0,blend_radius_m)
    |   movel([-0.046149, -1.398798, -2.562748, -0.750843, 1.570796, 1.524647],accel_mss,speed_ms,0,blend_radius_m)
    |   movel([-0.045182, -1.398133, -2.563233, -0.751022, 1.570796, 1.525614],accel_mss,speed_ms,0,blend_radius_m)
    |   movel([-0.044274, -1.397659, -2.563579, -0.751151, 1.570796, 1.526522],accel_mss,speed_ms,0,blend_radius_m)
    |   movel([-0.043471, -1.397443, -2.563737, -0.751209, 1.570796, 1.527325],accel_mss,speed_ms,0,blend_radius_m)
    |   movel([-0.042803, -1.397569, -2.563645, -0.751175, 1.570796, 1.527993],accel_mss,speed_ms,0,blend_radius_m)
    |   movel([-0.042348, -1.398020, -2.563316, -0.751053, 1.570796, 1.528448],accel_mss,speed_ms,0,blend_radius_m)
    |   movel([-0.042088, -1.398712, -2.562811, -0.750866, 1.570796, 1.528709],accel_mss,speed_ms,0,blend_radius_m)
    |   movel([-0.042011, -1.399560, -2.562190, -0.750639, 1.570796, 1.528786],accel_mss,speed_ms,0,blend_radius_m)
    |   movel([-0.042101, -1.400480, -2.561516, -0.750393, 1.570796, 1.528695],accel_mss,speed_ms,0,blend_radius_m)
    |   movel([-0.042343, -1.401386, -2.560851, -0.750152, 1.570796, 1.528454],accel_mss,speed_ms,0,blend_radius_m)
    |   movel([-0.042722, -1.402197, -2.560255, -0.749938, 1.570796, 1.528075],accel_mss,speed_ms,0,blend_radius_m)
    |   movel([-0.043225, -1.402828, -2.559790, -0.749771, 1.570796, 1.527572],accel_mss,speed_ms,0,blend_radius_m)
    |   movel([-0.040166, -1.400250, -2.561685, -0.750454, 1.570796, 1.530630],accel_mss,speed_ms,0,blend_radius_m)
    |   movel([-0.038546, -1.399062, -2.562555, -0.750772, 1.570796, 1.532251],accel_mss,speed_ms,0,blend_radius_m)
    |   movel([-0.036872, -1.397960, -2.563360, -0.751069, 1.570796, 1.533924],accel_mss,speed_ms,0,blend_radius_m)
    |   movel([-0.035156, -1.396957, -2.564091, -0.751341, 1.570796, 1.535640],accel_mss,speed_ms,0,blend_radius_m)
    |   movel([-0.033403, -1.396067, -2.564739, -0.751583, 1.570796, 1.537394],accel_mss,speed_ms,0,blend_radius_m)
    |   movel([-0.031619, -1.395304, -2.565293, -0.751792, 1.570796, 1.539177],accel_mss,speed_ms,0,blend_radius_m)
    |   movel([-0.029813, -1.394680, -2.565746, -0.751963, 1.570796, 1.540983],accel_mss,speed_ms,0,blend_radius_m)
    |   movel([-0.028597, -1.394494, -2.565881, -0.752015, 1.570796, 1.542199],accel_mss,speed_ms,0,blend_radius_m)
    |   movel([-0.027308, -1.394611, -2.565796, -0.751982, 1.570796, 1.543488],accel_mss,speed_ms,0,blend_radius_m)
    |   movel([-0.026754, -1.394802, -2.565657, -0.751930, 1.570796, 1.544042],accel_mss,speed_ms,0,blend_radius_m)
    |   movel([-0.026320, -1.395091, -2.565448, -0.751851, 1.570796, 1.544476],accel_mss,speed_ms,0,blend_radius_m)
    |   movel([-0.026051, -1.395484, -2.565162, -0.751743, 1.570796, 1.544745],accel_mss,speed_ms,0,blend_radius_m)
    |   movel([-0.025998, -1.395992, -2.564793, -0.751604, 1.570796, 1.544799],accel_mss,speed_ms,0,blend_radius_m)
    |   movel([-0.026188, -1.396540, -2.564395, -0.751454, 1.570796, 1.544608],accel_mss,speed_ms,0,blend_radius_m)
    |   movel([-0.026559, -1.397086, -2.563997, -0.751306, 1.570796, 1.544238],accel_mss,speed_ms,0,blend_radius_m)
    |   movel([-0.027646, -1.398202, -2.563183, -0.751004, 1.570796, 1.543150],accel_mss,speed_ms,0,blend_radius_m)
    |   movel([-0.028935, -1.399131, -2.562504, -0.750754, 1.570796, 1.541861],accel_mss,speed_ms,0,blend_radius_m)
    |   movel([-0.030340, -1.399897, -2.561943, -0.750548, 1.570796, 1.540456],accel_mss,speed_ms,0,blend_radius_m)
    |   movel([-0.031777, -1.400524, -2.561484, -0.750381, 1.570796, 1.539020],accel_mss,speed_ms,0,blend_radius_m)
    |   movel([-0.029959, -1.400609, -2.561422, -0.750359, 1.570796, 1.540838],accel_mss,speed_ms,0,blend_radius_m)
    |   movel([-0.028062, -1.400516, -2.561490, -0.750383, 1.570796, 1.542735],accel_mss,speed_ms,0,blend_radius_m)
    |   movel([-0.026107, -1.400250, -2.561685, -0.750454, 1.570796, 1.544690],accel_mss,speed_ms,0,blend_radius_m)
    |   movel([-0.024112, -1.399814, -2.562004, -0.750571, 1.570796, 1.546684],accel_mss,speed_ms,0,blend_radius_m)
    |   movel([-0.022533, -1.399314, -2.562370, -0.750705, 1.570796, 1.548263],accel_mss,speed_ms,0,blend_radius_m)
    |   movel([-0.019437, -1.398102, -2.563256, -0.751031, 1.570796, 1.551359],accel_mss,speed_ms,0,blend_radius_m)
    |   movel([-0.017855, -1.397589, -2.563630, -0.751169, 1.570796, 1.552941],accel_mss,speed_ms,0,blend_radius_m)
    |   movel([-0.016060, -1.397130, -2.563965, -0.751294, 1.570796, 1.554737],accel_mss,speed_ms,0,blend_radius_m)
    |   movel([-0.013047, -1.396511, -2.564416, -0.751462, 1.570796, 1.557749],accel_mss,speed_ms,0,blend_radius_m)
    |   movel([-0.011613, -1.396336, -2.564543, -0.751510, 1.570796, 1.559183],accel_mss,speed_ms,0,blend_radius_m)
    |   movel([-0.010507, -1.396353, -2.564531, -0.751505, 1.570796, 1.560289],accel_mss,speed_ms,0,blend_radius_m)
    |   movel([-0.010142, -1.396457, -2.564455, -0.751477, 1.570796, 1.560654],accel_mss,speed_ms,0,blend_radius_m)
    |   movel([-0.009941, -1.396639, -2.564322, -0.751427, 1.570796, 1.560855],accel_mss,speed_ms,0,blend_radius_m)
    |   movel([-0.009926, -1.396905, -2.564129, -0.751355, 1.570796, 1.560871],accel_mss,speed_ms,0,blend_radius_m)
    |   movel([-0.010125, -1.397265, -2.563866, -0.751257, 1.570796, 1.560671],accel_mss,speed_ms,0,blend_radius_m)
    |   movel([-0.010875, -1.398064, -2.563284, -0.751041, 1.570796, 1.559921],accel_mss,speed_ms,0,blend_radius_m)
    |   movel([-0.011846, -1.398827, -2.562726, -0.750835, 1.570796, 1.558951],accel_mss,speed_ms,0,blend_radius_m)
    |   movel([-0.012974, -1.399552, -2.562196, -0.750641, 1.570796, 1.557822],accel_mss,speed_ms,0,blend_radius_m)
    |   movel([-0.014194, -1.400229, -2.561700, -0.750460, 1.570796, 1.556602],accel_mss,speed_ms,0,blend_radius_m)
    |   movel([-0.016663, -1.401417, -2.560828, -0.750144, 1.570796, 1.554134],accel_mss,speed_ms,0,blend_radius_m)
    |   movel([-0.018743, -1.402340, -2.560149, -0.749900, 1.570796, 1.552053],accel_mss,speed_ms,0,blend_radius_m)
    |   movel([-0.017712, -1.402591, -2.559964, -0.749834, 1.570796, 1.553085],accel_mss,speed_ms,0,blend_radius_m)
    |   movel([-0.016621, -1.402742, -2.559853, -0.749794, 1.570796, 1.554176],accel_mss,speed_ms,0,blend_radius_m)
    |   movel([-0.014303, -1.402794, -2.559815, -0.749780, 1.570796, 1.556493],accel_mss,speed_ms,0,blend_radius_m)
    |   movel([-0.011861, -1.402587, -2.559967, -0.749835, 1.570796, 1.558936],accel_mss,speed_ms,0,blend_radius_m)
    |   movel([-0.009363, -1.402213, -2.560243, -0.749933, 1.570796, 1.561434],accel_mss,speed_ms,0,blend_radius_m)
    |   movel([-0.007287, -1.401786, -2.560557, -0.750046, 1.570796, 1.563509],accel_mss,speed_ms,0,blend_radius_m)
    |   movel([-0.001019, -1.400276, -2.561666, -0.750447, 1.570796, 1.569778],accel_mss,speed_ms,0,blend_radius_m)
    |   movel([0.000136, -1.400180, -2.561736, -0.750473, 1.570796, 1.570932],accel_mss,speed_ms,0,blend_radius_m)
    |   movel([0.001035, -1.400358, -2.561606, -0.750426, 1.570796, 1.571832],accel_mss,speed_ms,0,blend_radius_m)
    |   movel([0.001220, -1.400571, -2.561450, -0.750369, 1.570796, 1.572016],accel_mss,speed_ms,0,blend_radius_m)
    |   movel([0.001136, -1.400879, -2.561224, -0.750287, 1.570796, 1.571932],accel_mss,speed_ms,0,blend_radius_m)
    |   movel([0.000714, -1.401289, -2.560922, -0.750178, 1.570796, 1.571510],accel_mss,speed_ms,0,blend_radius_m)
    |   movel([-0.000113, -1.401810, -2.560539, -0.750040, 1.570796, 1.570683],accel_mss,speed_ms,0,blend_radius_m)
    |   movel([-0.001501, -1.402493, -2.560036, -0.749859, 1.570796, 1.569296],accel_mss,speed_ms,0,blend_radius_m)
    |   movel([-0.003103, -1.403126, -2.559570, -0.749693, 1.570796, 1.567693],accel_mss,speed_ms,0,blend_radius_m)
    |   movel([-0.004684, -1.403568, -2.559244, -0.749577, 1.570796, 1.566113],accel_mss,speed_ms,0,blend_radius_m)
    |   movel([-0.005392, -1.403675, -2.559165, -0.749549, 1.570796, 1.565405],accel_mss,speed_ms,0,blend_radius_m)
    |   movel([-0.006002, -1.403679, -2.559162, -0.749548, 1.570796, 1.564794],accel_mss,speed_ms,0,blend_radius_m)
    |   movel([-0.003636, -1.404544, -2.558523, -0.749322, 1.570796, 1.567160],accel_mss,speed_ms,0,blend_radius_m)
    |   movel([-0.001096, -1.405162, -2.558066, -0.749161, 1.570796, 1.569700],accel_mss,speed_ms,0,blend_radius_m)
    |   movel([0.001580, -1.405578, -2.557757, -0.749053, 1.570796, 1.572376],accel_mss,speed_ms,0,blend_radius_m)
    |   movel([0.004358, -1.405841, -2.557562, -0.748985, 1.570796, 1.575155],accel_mss,speed_ms,0,blend_radius_m)
    |   movel([0.010072, -1.406085, -2.557382, -0.748922, 1.570796, 1.580868],accel_mss,speed_ms,0,blend_radius_m)
    |   movel([0.015745, -1.406260, -2.557252, -0.748877, 1.570796, 1.586542],accel_mss,speed_ms,0,blend_radius_m)
    |   movel([0.016685, -1.406434, -2.557122, -0.748832, 1.570796, 1.587482],accel_mss,speed_ms,0,blend_radius_m)
    |   movel([0.016994, -1.406671, -2.556947, -0.748771, 1.570796, 1.587790],accel_mss,speed_ms,0,blend_radius_m)
    |   movel([0.017081, -1.407052, -2.556663, -0.748673, 1.570796, 1.587877],accel_mss,speed_ms,0,blend_radius_m)
    |   movel([0.016911, -1.407502, -2.556329, -0.748558, 1.570796, 1.587708],accel_mss,speed_ms,0,blend_radius_m)
    |   movel([0.015985, -1.408575, -2.555530, -0.748284, 1.570796, 1.586781],accel_mss,speed_ms,0,blend_radius_m)
    |   movel([0.015320, -1.409142, -2.555107, -0.748140, 1.570796, 1.586116],accel_mss,speed_ms,0,blend_radius_m)
    |   movel([0.013817, -1.410100, -2.554391, -0.747897, 1.570796, 1.584614],accel_mss,speed_ms,0,blend_radius_m)
    |   movel([0.012159, -1.410835, -2.553841, -0.747712, 1.570796, 1.582955],accel_mss,speed_ms,0,blend_radius_m)
    |   movel([0.010414, -1.411373, -2.553438, -0.747578, 1.570796, 1.581211],accel_mss,speed_ms,0,blend_radius_m)
    |   movel([0.008663, -1.411731, -2.553170, -0.747488, 1.570796, 1.579460],accel_mss,speed_ms,0,blend_radius_m)
    |   movel([0.006980, -1.411932, -2.553019, -0.747438, 1.570796, 1.577776],accel_mss,speed_ms,0,blend_radius_m)
    |   movel([0.005437, -1.411996, -2.552971, -0.747422, 1.570796, 1.576233],accel_mss,speed_ms,0,blend_radius_m)
    |   movel([0.004115, -1.411939, -2.553014, -0.747436, 1.570796, 1.574911],accel_mss,speed_ms,0,blend_radius_m)
    |   movel([0.004101, -1.412306, -2.552739, -0.747345, 1.570796, 1.574897],accel_mss,speed_ms,0,blend_radius_m)
    |   movel([0.004332, -1.412571, -2.552539, -0.747279, 1.570796, 1.575129],accel_mss,speed_ms,0,blend_radius_m)
    |   movel([0.005050, -1.413018, -2.552204, -0.747168, 1.570796, 1.575846],accel_mss,speed_ms,0,blend_radius_m)
    |   movel([0.005864, -1.413355, -2.551950, -0.747084, 1.570796, 1.576660],accel_mss,speed_ms,0,blend_radius_m)
    |   movel([0.007653, -1.413832, -2.551590, -0.746966, 1.570796, 1.578449],accel_mss,speed_ms,0,blend_radius_m)
    |   movel([0.010843, -1.414489, -2.551095, -0.746805, 1.570796, 1.581640],accel_mss,speed_ms,0,blend_radius_m)
    |   movel([0.014087, -1.415030, -2.550687, -0.746672, 1.570796, 1.584883],accel_mss,speed_ms,0,blend_radius_m)
    |   movel([0.020731, -1.415822, -2.550089, -0.746479, 1.570796, 1.591527],accel_mss,speed_ms,0,blend_radius_m)
    |   movel([0.022573, -1.416072, -2.549899, -0.746418, 1.570796, 1.593369],accel_mss,speed_ms,0,blend_radius_m)
    |   movel([0.023740, -1.416328, -2.549705, -0.746355, 1.570796, 1.594536],accel_mss,speed_ms,0,blend_radius_m)
    |   movel([0.024859, -1.416697, -2.549426, -0.746266, 1.570796, 1.595655],accel_mss,speed_ms,0,blend_radius_m)
    |   movel([0.025765, -1.417197, -2.549047, -0.746145, 1.570796, 1.596561],accel_mss,speed_ms,0,blend_radius_m)
    |   movel([0.026296, -1.417842, -2.548558, -0.745989, 1.570796, 1.597093],accel_mss,speed_ms,0,blend_radius_m)
    |   movel([0.026375, -1.418223, -2.548269, -0.745898, 1.570796, 1.597171],accel_mss,speed_ms,0,blend_radius_m)
    |   movel([0.026302, -1.418647, -2.547946, -0.745796, 1.570796, 1.597098],accel_mss,speed_ms,0,blend_radius_m)
    |   movel([0.026053, -1.419117, -2.547588, -0.745684, 1.570796, 1.596850],accel_mss,speed_ms,0,blend_radius_m)
    |   movel([0.025615, -1.419633, -2.547196, -0.745561, 1.570796, 1.596412],accel_mss,speed_ms,0,blend_radius_m)
    |   movel([0.024960, -1.420017, -2.546903, -0.745469, 1.570796, 1.595756],accel_mss,speed_ms,0,blend_radius_m)
    |   movel([0.024058, -1.420281, -2.546701, -0.745407, 1.570796, 1.594855],accel_mss,speed_ms,0,blend_radius_m)
    |   movel([0.019204, -1.421203, -2.545998, -0.745189, 1.570796, 1.590000],accel_mss,speed_ms,0,blend_radius_m)
    |   movel([0.017567, -1.421316, -2.545911, -0.745162, 1.570796, 1.588363],accel_mss,speed_ms,0,blend_radius_m)
    |   movel([0.016862, -1.421258, -2.545955, -0.745176, 1.570796, 1.587658],accel_mss,speed_ms,0,blend_radius_m)
    |   movel([0.016278, -1.421094, -2.546081, -0.745214, 1.570796, 1.587074],accel_mss,speed_ms,0,blend_radius_m)
    |   movel([0.018723, -1.422630, -2.544905, -0.744854, 1.570796, 1.589519],accel_mss,speed_ms,0,blend_radius_m)
    |   movel([0.021438, -1.423860, -2.543961, -0.744568, 1.570796, 1.592234],accel_mss,speed_ms,0,blend_radius_m)
    |   movel([0.024358, -1.424834, -2.543212, -0.744343, 1.570796, 1.595154],accel_mss,speed_ms,0,blend_radius_m)
    |   movel([0.027421, -1.425597, -2.542624, -0.744168, 1.570796, 1.598218],accel_mss,speed_ms,0,blend_radius_m)
    |   movel([0.030058, -1.425902, -2.542389, -0.744098, 1.570796, 1.600854],accel_mss,speed_ms,0,blend_radius_m)
    |   movel([0.033837, -1.426402, -2.542003, -0.743984, 1.570796, 1.604633],accel_mss,speed_ms,0,blend_radius_m)
    |   movel([0.035556, -1.426815, -2.541684, -0.743890, 1.570796, 1.606352],accel_mss,speed_ms,0,blend_radius_m)
    |   movel([0.036847, -1.427381, -2.541247, -0.743762, 1.570796, 1.607643],accel_mss,speed_ms,0,blend_radius_m)
    |   movel([0.037257, -1.427731, -2.540975, -0.743682, 1.570796, 1.608053],accel_mss,speed_ms,0,blend_radius_m)
    |   movel([0.037469, -1.428131, -2.540666, -0.743592, 1.570796, 1.608265],accel_mss,speed_ms,0,blend_radius_m)
    |   movel([0.037455, -1.428587, -2.540312, -0.743490, 1.570796, 1.608252],accel_mss,speed_ms,0,blend_radius_m)
    |   movel([0.037191, -1.429098, -2.539915, -0.743375, 1.570796, 1.607987],accel_mss,speed_ms,0,blend_radius_m)
    |   movel([0.036771, -1.429574, -2.539546, -0.743269, 1.570796, 1.607567],accel_mss,speed_ms,0,blend_radius_m)
    |   movel([0.036278, -1.429998, -2.539217, -0.743174, 1.570796, 1.607075],accel_mss,speed_ms,0,blend_radius_m)
    |   movel([0.035178, -1.430727, -2.538649, -0.743013, 1.570796, 1.605975],accel_mss,speed_ms,0,blend_radius_m)
    |   movel([0.033953, -1.431402, -2.538124, -0.742864, 1.570796, 1.604749],accel_mss,speed_ms,0,blend_radius_m)
    |   movel([0.031448, -1.432496, -2.537270, -0.742624, 1.570796, 1.602244],accel_mss,speed_ms,0,blend_radius_m)
    |   movel([0.030184, -1.432911, -2.536945, -0.742533, 1.570796, 1.600981],accel_mss,speed_ms,0,blend_radius_m)
    |   movel([0.032542, -1.433431, -2.536538, -0.742420, 1.570796, 1.603338],accel_mss,speed_ms,0,blend_radius_m)
    |   movel([0.034969, -1.433808, -2.536243, -0.742338, 1.570796, 1.605765],accel_mss,speed_ms,0,blend_radius_m)
    |   movel([0.037457, -1.434060, -2.536045, -0.742284, 1.570796, 1.608253],accel_mss,speed_ms,0,blend_radius_m)
    |   movel([0.040000, -1.434199, -2.535936, -0.742253, 1.570796, 1.610797],accel_mss,speed_ms,0,blend_radius_m)
    |   movel([0.045221, -1.434207, -2.535930, -0.742252, 1.570796, 1.616017],accel_mss,speed_ms,0,blend_radius_m)
    |   movel([0.050575, -1.433945, -2.536136, -0.742309, 1.570796, 1.621371],accel_mss,speed_ms,0,blend_radius_m)
    |   movel([0.051984, -1.434006, -2.536088, -0.742295, 1.570796, 1.622781],accel_mss,speed_ms,0,blend_radius_m)
    |   movel([0.052501, -1.434244, -2.535901, -0.742244, 1.570796, 1.623297],accel_mss,speed_ms,0,blend_radius_m)
    |   movel([0.052736, -1.434706, -2.535539, -0.742144, 1.570796, 1.623532],accel_mss,speed_ms,0,blend_radius_m)
    |   movel([0.052700, -1.435095, -2.535234, -0.742061, 1.570796, 1.623496],accel_mss,speed_ms,0,blend_radius_m)
    |   movel([0.052533, -1.435492, -2.534921, -0.741975, 1.570796, 1.623330],accel_mss,speed_ms,0,blend_radius_m)
    |   movel([0.051867, -1.436310, -2.534278, -0.741801, 1.570796, 1.622663],accel_mss,speed_ms,0,blend_radius_m)
    |   movel([0.050864, -1.437120, -2.533640, -0.741629, 1.570796, 1.621660],accel_mss,speed_ms,0,blend_radius_m)
    |   movel([0.049650, -1.437891, -2.533032, -0.741467, 1.570796, 1.620446],accel_mss,speed_ms,0,blend_radius_m)
    |   movel([0.047098, -1.439176, -2.532015, -0.741197, 1.570796, 1.617895],accel_mss,speed_ms,0,blend_radius_m)
    |   movel([0.045218, -1.439885, -2.531454, -0.741050, 1.570796, 1.616015],accel_mss,speed_ms,0,blend_radius_m)
    |   movel([0.046303, -1.439936, -2.531413, -0.741039, 1.570796, 1.617099],accel_mss,speed_ms,0,blend_radius_m)
    |   movel([0.047423, -1.439889, -2.531451, -0.741049, 1.570796, 1.618219],accel_mss,speed_ms,0,blend_radius_m)
    |   movel([0.049742, -1.439530, -2.531735, -0.741124, 1.570796, 1.620538],accel_mss,speed_ms,0,blend_radius_m)
    |   movel([0.052127, -1.438842, -2.532280, -0.741267, 1.570796, 1.622924],accel_mss,speed_ms,0,blend_radius_m)
    |   movel([0.054533, -1.437867, -2.533050, -0.741472, 1.570796, 1.625330],accel_mss,speed_ms,0,blend_radius_m)
    |   movel([0.056914, -1.436636, -2.534021, -0.741732, 1.570796, 1.627711],accel_mss,speed_ms,0,blend_radius_m)
    |   movel([0.059223, -1.435192, -2.535157, -0.742040, 1.570796, 1.630019],accel_mss,speed_ms,0,blend_radius_m)
    |   movel([0.061412, -1.433566, -2.536433, -0.742391, 1.570796, 1.632208],accel_mss,speed_ms,0,blend_radius_m)
    |   movel([0.063435, -1.431798, -2.537814, -0.742777, 1.570796, 1.634231],accel_mss,speed_ms,0,blend_radius_m)
    |   movel([0.064325, -1.431007, -2.538431, -0.742951, 1.570796, 1.635121],accel_mss,speed_ms,0,blend_radius_m)
    |   movel([0.064810, -1.430692, -2.538676, -0.743020, 1.570796, 1.635607],accel_mss,speed_ms,0,blend_radius_m)
    |   movel([0.065322, -1.430491, -2.538833, -0.743065, 1.570796, 1.636119],accel_mss,speed_ms,0,blend_radius_m)
    |   movel([0.065860, -1.430459, -2.538858, -0.743072, 1.570796, 1.636657],accel_mss,speed_ms,0,blend_radius_m)
    |   movel([0.066324, -1.430583, -2.538762, -0.743045, 1.570796, 1.637120],accel_mss,speed_ms,0,blend_radius_m)
    |   movel([0.066842, -1.431005, -2.538433, -0.742951, 1.570796, 1.637638],accel_mss,speed_ms,0,blend_radius_m)
    |   movel([0.067132, -1.431666, -2.537918, -0.742806, 1.570796, 1.637928],accel_mss,speed_ms,0,blend_radius_m)
    |   movel([0.067232, -1.432498, -2.537267, -0.742623, 1.570796, 1.638028],accel_mss,speed_ms,0,blend_radius_m)
    |   movel([0.067182, -1.433445, -2.536527, -0.742417, 1.570796, 1.637978],accel_mss,speed_ms,0,blend_radius_m)
    |   movel([0.066780, -1.435417, -2.534981, -0.741992, 1.570796, 1.637576],accel_mss,speed_ms,0,blend_radius_m)
    |   movel([0.066238, -1.437082, -2.533670, -0.741637, 1.570796, 1.637035],accel_mss,speed_ms,0,blend_radius_m)
    |   movel([0.067950, -1.435277, -2.535090, -0.742022, 1.570796, 1.638746],accel_mss,speed_ms,0,blend_radius_m)
    |   movel([0.069463, -1.433379, -2.536579, -0.742431, 1.570796, 1.640260],accel_mss,speed_ms,0,blend_radius_m)
    |   movel([0.070769, -1.431410, -2.538117, -0.742862, 1.570796, 1.641565],accel_mss,speed_ms,0,blend_radius_m)
    |   movel([0.071860, -1.429398, -2.539683, -0.743308, 1.570796, 1.642657],accel_mss,speed_ms,0,blend_radius_m)
    |   movel([0.072723, -1.427369, -2.541256, -0.743764, 1.570796, 1.643520],accel_mss,speed_ms,0,blend_radius_m)
    |   movel([0.073356, -1.425347, -2.542817, -0.744225, 1.570796, 1.644153],accel_mss,speed_ms,0,blend_radius_m)
    |   movel([0.073744, -1.423362, -2.544343, -0.744683, 1.570796, 1.644540],accel_mss,speed_ms,0,blend_radius_m)
    |   movel([0.073879, -1.421440, -2.545816, -0.745133, 1.570796, 1.644675],accel_mss,speed_ms,0,blend_radius_m)
    |   movel([0.073661, -1.418892, -2.547760, -0.745737, 1.570796, 1.644458],accel_mss,speed_ms,0,blend_radius_m)
    |   movel([0.073663, -1.417520, -2.548802, -0.746067, 1.570796, 1.644460],accel_mss,speed_ms,0,blend_radius_m)
    |   movel([0.073776, -1.416854, -2.549307, -0.746228, 1.570796, 1.644572],accel_mss,speed_ms,0,blend_radius_m)
    |   movel([0.073991, -1.416217, -2.549790, -0.746382, 1.570796, 1.644787],accel_mss,speed_ms,0,blend_radius_m)
    |   movel([0.074550, -1.415234, -2.550533, -0.746622, 1.570796, 1.645347],accel_mss,speed_ms,0,blend_radius_m)
    |   movel([0.075106, -1.414698, -2.550937, -0.746753, 1.570796, 1.645903],accel_mss,speed_ms,0,blend_radius_m)
    |   movel([0.075657, -1.414513, -2.551077, -0.746799, 1.570796, 1.646454],accel_mss,speed_ms,0,blend_radius_m)
    |   movel([0.076198, -1.414581, -2.551026, -0.746782, 1.570796, 1.646994],accel_mss,speed_ms,0,blend_radius_m)
    |   movel([0.077684, -1.415340, -2.550453, -0.746596, 1.570796, 1.648480],accel_mss,speed_ms,0,blend_radius_m)
    |   movel([0.078118, -1.415453, -2.550367, -0.746569, 1.570796, 1.648914],accel_mss,speed_ms,0,blend_radius_m)
    |   movel([0.078894, -1.413988, -2.551473, -0.746928, 1.570796, 1.649690],accel_mss,speed_ms,0,blend_radius_m)
    |   movel([0.079523, -1.412498, -2.552594, -0.747297, 1.570796, 1.650319],accel_mss,speed_ms,0,blend_radius_m)
    |   movel([0.080014, -1.410991, -2.553724, -0.747673, 1.570796, 1.650810],accel_mss,speed_ms,0,blend_radius_m)
    |   movel([0.080375, -1.409474, -2.554859, -0.748056, 1.570796, 1.651171],accel_mss,speed_ms,0,blend_radius_m)
    |   movel([0.080608, -1.407958, -2.555990, -0.748441, 1.570796, 1.651405],accel_mss,speed_ms,0,blend_radius_m)
    |   movel([0.080723, -1.406448, -2.557113, -0.748829, 1.570796, 1.651520],accel_mss,speed_ms,0,blend_radius_m)
    |   movel([0.080635, -1.403476, -2.559312, -0.749601, 1.570796, 1.651431],accel_mss,speed_ms,0,blend_radius_m)
    |   movel([0.080162, -1.400629, -2.561407, -0.750353, 1.570796, 1.650958],accel_mss,speed_ms,0,blend_radius_m)
    |   movel([0.079372, -1.397967, -2.563355, -0.751067, 1.570796, 1.650169],accel_mss,speed_ms,0,blend_radius_m)
    |   movel([0.078320, -1.395559, -2.565108, -0.751722, 1.570796, 1.649116],accel_mss,speed_ms,0,blend_radius_m)
    |   movel([0.077075, -1.393466, -2.566625, -0.752298, 1.570796, 1.647871],accel_mss,speed_ms,0,blend_radius_m)
    |   speed_ms = 0.005
    |   movel([0.077075, -1.384778, -2.562689, -0.764923, 1.570796, 1.647871],accel_mss,speed_ms,0,blend_radius_m)
    |   speed_ms = 0.040
    |   movel([0.063534, -1.389965, -2.558967, -0.763456, 1.570796, 1.634331],accel_mss,speed_ms,0,blend_radius_m)
    |   speed_ms = 0.005
    |   movel([0.063534, -1.398616, -2.562881, -0.750892, 1.570796, 1.634331],accel_mss,speed_ms,0,blend_radius_m)
    |   speed_ms = 0.025
    |   movel([0.062308, -1.398046, -2.563297, -0.751046, 1.570796, 1.633105],accel_mss,speed_ms,0,blend_radius_m)
    |   movel([0.060907, -1.397768, -2.563500, -0.751121, 1.570796, 1.631703],accel_mss,speed_ms,0,blend_radius_m)
